ABB RAPID module: Module1.mod

MODULE Module1

     VAR robtarget current_position;
     VAR robtarget starting_position;
     VAR jointtarget joints;
    TASK PERS wobjdata wobj:=[FALSE,FALSE,"ROB_1",[[639.116,-22.796,-980.437],[1,0,0,0]],[[0,0,0],[1,0,0,0]]];

    PROC main()

starting_position := CRobT(\TaskName:="T_ROB1" \Tool:=Tooldata_9);
MoveJ RelTool (starting_position, 342,4, -480.2 \Rx:=7.6, \Ry:=21.9, \Rz:=1), v200, z200, Tooldata_9;
MoveJ RelTool (starting_position, 341,4, -481.5 \Rx:=7.6, \Ry:=21.6, \Rz:=1), v200, z200, Tooldata_9;
MoveJ RelTool (starting_position, 339,4, -483.2 \Rx:=7.6, \Ry:=21.6, \Rz:=1), v200, z200, Tooldata_9;
MoveJ RelTool (starting_position, 338,4, -485.4 \Rx:=7.5, \Ry:=21.3, \Rz:=1), v200, z200, Tooldata_9;
MoveJ RelTool (starting_position, 336,4, -488.1 \Rx:=7.5, \Ry:=21.3, \Rz:=1), v200, z200, Tooldata_9;
MoveJ RelTool (starting_position, 334,4, -491.4 \Rx:=7.5, \Ry:=21, \Rz:=1), v200, z200, Tooldata_9;
MoveJ RelTool (starting_position, 332,4, -495.2 \Rx:=7.5, \Ry:=20.7, \Rz:=1), v200, z200, Tooldata_9;
MoveJ RelTool (starting_position, 330,4, -499.5 \Rx:=7.5, \Ry:=20.4, \Rz:=1), v200, z200, Tooldata_9;
MoveJ RelTool (starting_position, 327,4, -504.2 \Rx:=7.5, \Ry:=20.1, \Rz:=1), v200, z200, Tooldata_9;
MoveJ RelTool (starting_position, 324,4, -509.1 \Rx:=7.5, \Ry:=19.8, \Rz:=1), v200, z200, Tooldata_9;
MoveJ RelTool (starting_position, 322,4, -514 \Rx:=7.6, \Ry:=19.5, \Rz:=1), v200, z200, Tooldata_9;
MoveJ RelTool (starting_position, 318,4, -518.8 \Rx:=7.6, \Ry:=19.5, \Rz:=1), v200, z200, Tooldata_9;
MoveJ RelTool (starting_position, 315,4, -523.4 \Rx:=7.6, \Ry:=19.2, \Rz:=1), v200, z200, Tooldata_9;
MoveJ RelTool (starting_position, 312,4, -527.5 \Rx:=7.6, \Ry:=18.9, \Rz:=1), v200, z200, Tooldata_9;
MoveJ RelTool (starting_position, 308,4, -531.3 \Rx:=7.6, \Ry:=18.6, \Rz:=1), v200, z200, Tooldata_9;
MoveJ RelTool (starting_position, 305,4, -534.7 \Rx:=7.6, \Ry:=18.3, \Rz:=1), v200, z200, Tooldata_9;
MoveJ RelTool (starting_position, 301,4, -537.8 \Rx:=7.6, \Ry:=18, \Rz:=1), v200, z200, Tooldata_9;
MoveJ RelTool (starting_position, 297,8, -540.6 \Rx:=7.6, \Ry:=17.4, \Rz:=2), v200, z200, Tooldata_9;
MoveJ RelTool (starting_position, 293,8, -543.1 \Rx:=7.6, \Ry:=17.1, \Rz:=2), v200, z200, Tooldata_9;
MoveJ RelTool (starting_position, 288,8, -545.5 \Rx:=7.6, \Ry:=16.8, \Rz:=2), v200, z200, Tooldata_9;
MoveJ RelTool (starting_position, 284,8, -547.8 \Rx:=7.6, \Ry:=16.5, \Rz:=2), v200, z200, Tooldata_9;
MoveJ RelTool (starting_position, 280,8, -550 \Rx:=7.6, \Ry:=15.9, \Rz:=2), v200, z200, Tooldata_9;
MoveJ RelTool (starting_position, 275,8, -552.2 \Rx:=7.6, \Ry:=15.6, \Rz:=2), v200, z200, Tooldata_9;
MoveJ RelTool (starting_position, 271,8, -554.4 \Rx:=7.6, \Ry:=15.3, \Rz:=2), v200, z200, Tooldata_9;
MoveJ RelTool (starting_position, 266,8, -556.6 \Rx:=7.7, \Ry:=14.7, \Rz:=2), v200, z200, Tooldata_9;
MoveJ RelTool (starting_position, 261,8, -558.8 \Rx:=7.7, \Ry:=14.4, \Rz:=2), v200, z200, Tooldata_9;
MoveJ RelTool (starting_position, 257,8, -561.1 \Rx:=7.7, \Ry:=14.1, \Rz:=2), v200, z200, Tooldata_9;
MoveJ RelTool (starting_position, 252,8, -563.3 \Rx:=7.7, \Ry:=13.5, \Rz:=2), v200, z200, Tooldata_9;
MoveJ RelTool (starting_position, 248,8, -565.6 \Rx:=7.7, \Ry:=13.2, \Rz:=2), v200, z200, Tooldata_9;
MoveJ RelTool (starting_position, 243,8, -567.8 \Rx:=7.7, \Ry:=12.9, \Rz:=2), v200, z200, Tooldata_9;
MoveJ RelTool (starting_position, 239,8, -570.1 \Rx:=7.7, \Ry:=12.3, \Rz:=2), v200, z200, Tooldata_9;
MoveJ RelTool (starting_position, 234,8, -572.3 \Rx:=7.7, \Ry:=12, \Rz:=2), v200, z200, Tooldata_9;
MoveJ RelTool (starting_position, 230,8, -574.4 \Rx:=7.7, \Ry:=11.7, \Rz:=2), v200, z200, Tooldata_9;
MoveJ RelTool (starting_position, 226,8, -576.4 \Rx:=7.7, \Ry:=11.4, \Rz:=2), v200, z200, Tooldata_9;
MoveJ RelTool (starting_position, 222,12, -578 \Rx:=7.8, \Ry:=10.8, \Rz:=3), v200, z200, Tooldata_9;
MoveJ RelTool (starting_position, 218,12, -579.3 \Rx:=7.8, \Ry:=10.5, \Rz:=3), v200, z200, Tooldata_9;
MoveJ RelTool (starting_position, 214,12, -580.4 \Rx:=7.8, \Ry:=10.2, \Rz:=3), v200, z200, Tooldata_9;
MoveJ RelTool (starting_position, 210,12, -581.1 \Rx:=7.8, \Ry:=9.9, \Rz:=3), v200, z200, Tooldata_9;
MoveJ RelTool (starting_position, 207,12, -581.4 \Rx:=7.8, \Ry:=9.6, \Rz:=3), v200, z200, Tooldata_9;
MoveJ RelTool (starting_position, 203,12, -581.5 \Rx:=7.8, \Ry:=9.3, \Rz:=3), v200, z200, Tooldata_9;
MoveJ RelTool (starting_position, 200,12, -581.3 \Rx:=7.8, \Ry:=9, \Rz:=3), v200, z200, Tooldata_9;
MoveJ RelTool (starting_position, 197,12, -580.9 \Rx:=7.8, \Ry:=8.7, \Rz:=3), v200, z200, Tooldata_9;
MoveJ RelTool (starting_position, 194,12, -580.4 \Rx:=7.8, \Ry:=8.4, \Rz:=3), v200, z200, Tooldata_9;
MoveJ RelTool (starting_position, 191,12, -579.7 \Rx:=7.8, \Ry:=8.4, \Rz:=3), v200, z200, Tooldata_9;
MoveJ RelTool (starting_position, 188,12, -579.2 \Rx:=7.8, \Ry:=8.1, \Rz:=3), v200, z200, Tooldata_9;
MoveJ RelTool (starting_position, 185,12, -578.8 \Rx:=7.8, \Ry:=7.8, \Rz:=3), v200, z200, Tooldata_9;
MoveJ RelTool (starting_position, 183,12, -578.9 \Rx:=7.8, \Ry:=7.5, \Rz:=3), v200, z200, Tooldata_9;
MoveJ RelTool (starting_position, 180,12, -579.4 \Rx:=7.8, \Ry:=7.2, \Rz:=3), v200, z200, Tooldata_9;
MoveJ RelTool (starting_position, 178,16, -580.4 \Rx:=7.8, \Ry:=7.2, \Rz:=4), v200, z200, Tooldata_9;
MoveJ RelTool (starting_position, 176,16, -582.1 \Rx:=7.8, \Ry:=6.9, \Rz:=4), v200, z200, Tooldata_9;
MoveJ RelTool (starting_position, 173,16, -584.3 \Rx:=7.8, \Ry:=6.9, \Rz:=4), v200, z200, Tooldata_9;
MoveJ RelTool (starting_position, 171,16, -587 \Rx:=7.8, \Ry:=6.6, \Rz:=4), v200, z200, Tooldata_9;
MoveJ RelTool (starting_position, 169,16, -589.9 \Rx:=7.8, \Ry:=6.3, \Rz:=4), v200, z200, Tooldata_9;
MoveJ RelTool (starting_position, 167,16, -592.9 \Rx:=7.8, \Ry:=6, \Rz:=4), v200, z200, Tooldata_9;
MoveJ RelTool (starting_position, 165,16, -595.7 \Rx:=7.7, \Ry:=6, \Rz:=4), v200, z200, Tooldata_9;
MoveJ RelTool (starting_position, 163,16, -598.3 \Rx:=7.7, \Ry:=6, \Rz:=4), v200, z200, Tooldata_9;
MoveJ RelTool (starting_position, 161,16, -600.4 \Rx:=7.7, \Ry:=5.7, \Rz:=4), v200, z200, Tooldata_9;
MoveJ RelTool (starting_position, 159,16, -602.1 \Rx:=7.7, \Ry:=5.4, \Rz:=4), v200, z200, Tooldata_9;
MoveJ RelTool (starting_position, 157,16, -603.5 \Rx:=7.7, \Ry:=5.4, \Rz:=4), v200, z200, Tooldata_9;
MoveJ RelTool (starting_position, 155,16, -604.4 \Rx:=7.6, \Ry:=5.1, \Rz:=4), v200, z200, Tooldata_9;
MoveJ RelTool (starting_position, 153,16, -605 \Rx:=7.6, \Ry:=5.1, \Rz:=4), v200, z200, Tooldata_9;
MoveJ RelTool (starting_position, 151,16, -605.4 \Rx:=7.6, \Ry:=4.8, \Rz:=4), v200, z200, Tooldata_9;
MoveJ RelTool (starting_position, 150,20, -605.6 \Rx:=7.5, \Ry:=4.8, \Rz:=5), v200, z200, Tooldata_9;
MoveJ RelTool (starting_position, 148,20, -605.7 \Rx:=7.5, \Ry:=4.5, \Rz:=5), v200, z200, Tooldata_9;
MoveJ RelTool (starting_position, 146,20, -605.8 \Rx:=7.5, \Ry:=4.5, \Rz:=5), v200, z200, Tooldata_9;
MoveJ RelTool (starting_position, 144,20, -605.8 \Rx:=7.4, \Ry:=4.2, \Rz:=5), v200, z200, Tooldata_9;
MoveJ RelTool (starting_position, 143,20, -605.8 \Rx:=7.4, \Ry:=4.2, \Rz:=5), v200, z200, Tooldata_9;
MoveJ RelTool (starting_position, 141,20, -605.8 \Rx:=7.3, \Ry:=3.9, \Rz:=5), v200, z200, Tooldata_9;
MoveJ RelTool (starting_position, 140,20, -605.8 \Rx:=7.3, \Ry:=3.9, \Rz:=5), v200, z200, Tooldata_9;
MoveJ RelTool (starting_position, 138,20, -605.8 \Rx:=7.2, \Ry:=3.6, \Rz:=5), v200, z200, Tooldata_9;
MoveJ RelTool (starting_position, 137,20, -605.8 \Rx:=7.2, \Ry:=3.6, \Rz:=5), v200, z200, Tooldata_9;
MoveJ RelTool (starting_position, 136,20, -605.8 \Rx:=7.1, \Ry:=3.6, \Rz:=5), v200, z200, Tooldata_9;
MoveJ RelTool (starting_position, 134,20, -605.8 \Rx:=7.1, \Ry:=3.3, \Rz:=5), v200, z200, Tooldata_9;
MoveJ RelTool (starting_position, 133,20, -605.8 \Rx:=7, \Ry:=3.3, \Rz:=5), v200, z200, Tooldata_9;
MoveJ RelTool (starting_position, 132,20, -605.8 \Rx:=6.9, \Ry:=3.3, \Rz:=5), v200, z200, Tooldata_9;
MoveJ RelTool (starting_position, 131,20, -605.8 \Rx:=6.9, \Ry:=3, \Rz:=5), v200, z200, Tooldata_9;
MoveJ RelTool (starting_position, 130,24, -605.8 \Rx:=6.8, \Ry:=3, \Rz:=6), v200, z200, Tooldata_9;
MoveJ RelTool (starting_position, 129,24, -605.8 \Rx:=6.7, \Ry:=3, \Rz:=6), v200, z200, Tooldata_9;
MoveJ RelTool (starting_position, 129,24, -605.8 \Rx:=6.7, \Ry:=3, \Rz:=6), v200, z200, Tooldata_9;
MoveJ RelTool (starting_position, 128,24, -605.8 \Rx:=6.6, \Ry:=2.7, \Rz:=6), v200, z200, Tooldata_9;
MoveJ RelTool (starting_position, 127,24, -606 \Rx:=6.5, \Ry:=2.7, \Rz:=6), v200, z200, Tooldata_9;
MoveJ RelTool (starting_position, 127,24, -606.4 \Rx:=6.4, \Ry:=2.7, \Rz:=6), v200, z200, Tooldata_9;
MoveJ RelTool (starting_position, 126,24, -606.9 \Rx:=6.3, \Ry:=2.7, \Rz:=6), v200, z200, Tooldata_9;
MoveJ RelTool (starting_position, 126,24, -607.5 \Rx:=6.2, \Ry:=2.7, \Rz:=6), v200, z200, Tooldata_9;
MoveJ RelTool (starting_position, 125,24, -608.2 \Rx:=6.2, \Ry:=2.7, \Rz:=6), v200, z200, Tooldata_9;
MoveJ RelTool (starting_position, 125,24, -609.1 \Rx:=6.1, \Ry:=2.7, \Rz:=6), v200, z200, Tooldata_9;
MoveJ RelTool (starting_position, 124,24, -610.2 \Rx:=6, \Ry:=2.7, \Rz:=6), v200, z200, Tooldata_9;
MoveJ RelTool (starting_position, 123,24, -611.3 \Rx:=5.9, \Ry:=2.4, \Rz:=6), v200, z200, Tooldata_9;
MoveJ RelTool (starting_position, 123,24, -612.3 \Rx:=5.8, \Ry:=2.4, \Rz:=6), v200, z200, Tooldata_9;
MoveJ RelTool (starting_position, 122,24, -613.3 \Rx:=5.7, \Ry:=2.4, \Rz:=6), v200, z200, Tooldata_9;
MoveJ RelTool (starting_position, 121,28, -614.1 \Rx:=5.7, \Ry:=2.4, \Rz:=7), v200, z200, Tooldata_9;
MoveJ RelTool (starting_position, 120,28, -614.8 \Rx:=5.6, \Ry:=2.1, \Rz:=7), v200, z200, Tooldata_9;
MoveJ RelTool (starting_position, 119,28, -615.4 \Rx:=5.5, \Ry:=2.1, \Rz:=7), v200, z200, Tooldata_9;
MoveJ RelTool (starting_position, 118,28, -616 \Rx:=5.4, \Ry:=2.1, \Rz:=7), v200, z200, Tooldata_9;
MoveJ RelTool (starting_position, 117,28, -616.7 \Rx:=5.3, \Ry:=1.8, \Rz:=7), v200, z200, Tooldata_9;
MoveJ RelTool (starting_position, 117,28, -617.3 \Rx:=5.3, \Ry:=1.8, \Rz:=7), v200, z200, Tooldata_9;
MoveJ RelTool (starting_position, 116,28, -618 \Rx:=5.2, \Ry:=1.8, \Rz:=7), v200, z200, Tooldata_9;
MoveJ RelTool (starting_position, 115,28, -618.7 \Rx:=5.1, \Ry:=1.8, \Rz:=7), v200, z200, Tooldata_9;
MoveJ RelTool (starting_position, 114,28, -619.2 \Rx:=5, \Ry:=1.8, \Rz:=7), v200, z200, Tooldata_9;
MoveJ RelTool (starting_position, 113,28, -619.6 \Rx:=4.9, \Ry:=1.5, \Rz:=7), v200, z200, Tooldata_9;
MoveJ RelTool (starting_position, 112,28, -619.8 \Rx:=4.8, \Ry:=1.5, \Rz:=7), v200, z200, Tooldata_9;
MoveJ RelTool (starting_position, 112,28, -619.9 \Rx:=4.7, \Ry:=1.5, \Rz:=7), v200, z200, Tooldata_9;
MoveJ RelTool (starting_position, 111,28, -619.8 \Rx:=4.6, \Ry:=1.5, \Rz:=7), v200, z200, Tooldata_9;
MoveJ RelTool (starting_position, 110,28, -619.5 \Rx:=4.5, \Ry:=1.2, \Rz:=7), v200, z200, Tooldata_9;
MoveJ RelTool (starting_position, 109,28, -619.2 \Rx:=4.4, \Ry:=1.2, \Rz:=7), v200, z200, Tooldata_9;
MoveJ RelTool (starting_position, 108,28, -618.8 \Rx:=4.4, \Ry:=1.2, \Rz:=7), v200, z200, Tooldata_9;
MoveJ RelTool (starting_position, 107,32, -618.4 \Rx:=4.3, \Ry:=1.2, \Rz:=8), v200, z200, Tooldata_9;
MoveJ RelTool (starting_position, 107,32, -618.2 \Rx:=4.2, \Ry:=0.9, \Rz:=8), v200, z200, Tooldata_9;
MoveJ RelTool (starting_position, 106,32, -618.1 \Rx:=4.1, \Ry:=0.9, \Rz:=8), v200, z200, Tooldata_9;
MoveJ RelTool (starting_position, 105,32, -618.2 \Rx:=4, \Ry:=0.9, \Rz:=8), v200, z200, Tooldata_9;
MoveJ RelTool (starting_position, 104,32, -618.4 \Rx:=3.9, \Ry:=0.9, \Rz:=8), v200, z200, Tooldata_9;
MoveJ RelTool (starting_position, 103,32, -618.8 \Rx:=3.8, \Ry:=0.6, \Rz:=8), v200, z200, Tooldata_9;
MoveJ RelTool (starting_position, 102,32, -619.2 \Rx:=3.7, \Ry:=0.6, \Rz:=8), v200, z200, Tooldata_9;
MoveJ RelTool (starting_position, 102,32, -619.7 \Rx:=3.6, \Ry:=0.6, \Rz:=8), v200, z200, Tooldata_9;
MoveJ RelTool (starting_position, 101,32, -620.1 \Rx:=3.6, \Ry:=0.6, \Rz:=8), v200, z200, Tooldata_9;
MoveJ RelTool (starting_position, 100,32, -620.4 \Rx:=3.5, \Ry:=0.6, \Rz:=8), v200, z200, Tooldata_9;
MoveJ RelTool (starting_position, 99,32, -620.7 \Rx:=3.4, \Ry:=0.3, \Rz:=8), v200, z200, Tooldata_9;
MoveJ RelTool (starting_position, 99,32, -620.8 \Rx:=3.3, \Ry:=0.3, \Rz:=8), v200, z200, Tooldata_9;
MoveJ RelTool (starting_position, 98,32, -620.9 \Rx:=3.2, \Ry:=0.3, \Rz:=8), v200, z200, Tooldata_9;
MoveJ RelTool (starting_position, 97,32, -620.9 \Rx:=3.2, \Ry:=0.3, \Rz:=8), v200, z200, Tooldata_9;
MoveJ RelTool (starting_position, 96,32, -620.7 \Rx:=3.1, \Ry:=0, \Rz:=8), v200, z200, Tooldata_9;
MoveJ RelTool (starting_position, 95,36, -620.5 \Rx:=3, \Ry:=0, \Rz:=9), v200, z200, Tooldata_9;
MoveJ RelTool (starting_position, 94,36, -620.2 \Rx:=2.9, \Ry:=-0, \Rz:=9), v200, z200, Tooldata_9;
MoveJ RelTool (starting_position, 94,36, -619.8 \Rx:=2.9, \Ry:=-0, \Rz:=9), v200, z200, Tooldata_9;
MoveJ RelTool (starting_position, 93,36, -619.4 \Rx:=2.8, \Ry:=-0.3, \Rz:=9), v200, z200, Tooldata_9;
MoveJ RelTool (starting_position, 92,36, -619 \Rx:=2.7, \Ry:=-0.3, \Rz:=9), v200, z200, Tooldata_9;
MoveJ RelTool (starting_position, 91,36, -618.5 \Rx:=2.7, \Ry:=-0.3, \Rz:=9), v200, z200, Tooldata_9;
MoveJ RelTool (starting_position, 90,36, -618.2 \Rx:=2.6, \Ry:=-0.3, \Rz:=9), v200, z200, Tooldata_9;
MoveJ RelTool (starting_position, 90,36, -617.9 \Rx:=2.5, \Ry:=-0.6, \Rz:=9), v200, z200, Tooldata_9;
MoveJ RelTool (starting_position, 89,36, -617.7 \Rx:=2.4, \Ry:=-0.6, \Rz:=9), v200, z200, Tooldata_9;
MoveJ RelTool (starting_position, 88,36, -617.7 \Rx:=2.4, \Ry:=-0.6, \Rz:=9), v200, z200, Tooldata_9;
MoveJ RelTool (starting_position, 87,36, -617.7 \Rx:=2.3, \Ry:=-0.6, \Rz:=9), v200, z200, Tooldata_9;
MoveJ RelTool (starting_position, 86,36, -617.8 \Rx:=2.2, \Ry:=-0.6, \Rz:=9), v200, z200, Tooldata_9;
MoveJ RelTool (starting_position, 85,36, -617.9 \Rx:=2.2, \Ry:=-0.6, \Rz:=9), v200, z200, Tooldata_9;
MoveJ RelTool (starting_position, 84,36, -618 \Rx:=2.1, \Ry:=-0.9, \Rz:=9), v200, z200, Tooldata_9;
MoveJ RelTool (starting_position, 83,36, -618.1 \Rx:=2, \Ry:=-0.9, \Rz:=9), v200, z200, Tooldata_9;
MoveJ RelTool (starting_position, 81,36, -618.1 \Rx:=1.9, \Ry:=-1.2, \Rz:=9), v200, z200, Tooldata_9;
MoveJ RelTool (starting_position, 80,36, -618.2 \Rx:=1.9, \Ry:=-1.2, \Rz:=9), v200, z200, Tooldata_9;
MoveJ RelTool (starting_position, 78,40, -618.2 \Rx:=1.8, \Ry:=-1.5, \Rz:=10), v200, z200, Tooldata_9;
MoveJ RelTool (starting_position, 77,40, -618.3 \Rx:=1.7, \Ry:=-1.5, \Rz:=10), v200, z200, Tooldata_9;
MoveJ RelTool (starting_position, 75,40, -618.3 \Rx:=1.7, \Ry:=-1.5, \Rz:=10), v200, z200, Tooldata_9;
MoveJ RelTool (starting_position, 73,40, -618.3 \Rx:=1.6, \Ry:=-1.8, \Rz:=10), v200, z200, Tooldata_9;
MoveJ RelTool (starting_position, 72,40, -618.3 \Rx:=1.6, \Ry:=-2.1, \Rz:=10), v200, z200, Tooldata_9;
MoveJ RelTool (starting_position, 70,40, -618.3 \Rx:=1.5, \Ry:=-2.1, \Rz:=10), v200, z200, Tooldata_9;
MoveJ RelTool (starting_position, 68,40, -618.3 \Rx:=1.4, \Ry:=-2.4, \Rz:=10), v200, z200, Tooldata_9;
MoveJ RelTool (starting_position, 66,40, -618.3 \Rx:=1.4, \Ry:=-2.4, \Rz:=10), v200, z200, Tooldata_9;
MoveJ RelTool (starting_position, 65,40, -618.3 \Rx:=1.3, \Ry:=-2.7, \Rz:=10), v200, z200, Tooldata_9;
MoveJ RelTool (starting_position, 63,40, -618.3 \Rx:=1.3, \Ry:=-2.7, \Rz:=10), v200, z200, Tooldata_9;
MoveJ RelTool (starting_position, 61,40, -618.3 \Rx:=1.2, \Ry:=-3, \Rz:=10), v200, z200, Tooldata_9;
MoveJ RelTool (starting_position, 59,40, -618.3 \Rx:=1.2, \Ry:=-3, \Rz:=10), v200, z200, Tooldata_9;
MoveJ RelTool (starting_position, 57,40, -618.3 \Rx:=1.1, \Ry:=-3.3, \Rz:=10), v200, z200, Tooldata_9;
MoveJ RelTool (starting_position, 56,40, -618.2 \Rx:=1.1, \Ry:=-3.3, \Rz:=10), v200, z200, Tooldata_9;
MoveJ RelTool (starting_position, 54,40, -618 \Rx:=1, \Ry:=-3.6, \Rz:=10), v200, z200, Tooldata_9;
MoveJ RelTool (starting_position, 52,40, -617.8 \Rx:=0.9, \Ry:=-3.6, \Rz:=10), v200, z200, Tooldata_9;
MoveJ RelTool (starting_position, 50,40, -617.3 \Rx:=0.9, \Ry:=-3.9, \Rz:=10), v200, z200, Tooldata_9;
MoveJ RelTool (starting_position, 49,40, -616.7 \Rx:=0.8, \Ry:=-4.2, \Rz:=10), v200, z200, Tooldata_9;
MoveJ RelTool (starting_position, 47,44, -615.8 \Rx:=0.8, \Ry:=-4.2, \Rz:=11), v200, z200, Tooldata_9;
MoveJ RelTool (starting_position, 46,44, -614.7 \Rx:=0.7, \Ry:=-4.2, \Rz:=11), v200, z200, Tooldata_9;
MoveJ RelTool (starting_position, 44,44, -613.4 \Rx:=0.7, \Ry:=-4.5, \Rz:=11), v200, z200, Tooldata_9;
MoveJ RelTool (starting_position, 43,44, -611.8 \Rx:=0.6, \Ry:=-4.5, \Rz:=11), v200, z200, Tooldata_9;
MoveJ RelTool (starting_position, 42,44, -610.2 \Rx:=0.5, \Ry:=-4.8, \Rz:=11), v200, z200, Tooldata_9;
MoveJ RelTool (starting_position, 41,44, -608.5 \Rx:=0.5, \Ry:=-4.8, \Rz:=11), v200, z200, Tooldata_9;
MoveJ RelTool (starting_position, 40,44, -607 \Rx:=0.4, \Ry:=-4.8, \Rz:=11), v200, z200, Tooldata_9;
MoveJ RelTool (starting_position, 39,44, -605.6 \Rx:=0.4, \Ry:=-4.8, \Rz:=11), v200, z200, Tooldata_9;
MoveJ RelTool (starting_position, 38,44, -604.4 \Rx:=0.3, \Ry:=-5.1, \Rz:=11), v200, z200, Tooldata_9;
MoveJ RelTool (starting_position, 38,44, -603.5 \Rx:=0.3, \Ry:=-5.1, \Rz:=11), v200, z200, Tooldata_9;
MoveJ RelTool (starting_position, 38,44, -602.9 \Rx:=0.2, \Ry:=-5.1, \Rz:=11), v200, z200, Tooldata_9;
MoveJ RelTool (starting_position, 38,44, -602.3 \Rx:=0.2, \Ry:=-5.1, \Rz:=11), v200, z200, Tooldata_9;
MoveJ RelTool (starting_position, 38,44, -601.9 \Rx:=0.1, \Ry:=-5.1, \Rz:=11), v200, z200, Tooldata_9;
MoveJ RelTool (starting_position, 38,44, -601.4 \Rx:=0.1, \Ry:=-5.1, \Rz:=11), v200, z200, Tooldata_9;
MoveJ RelTool (starting_position, 39,44, -600.8 \Rx:=0, \Ry:=-4.8, \Rz:=11), v200, z200, Tooldata_9;
MoveJ RelTool (starting_position, 40,44, -600.2 \Rx:=-0, \Ry:=-4.8, \Rz:=11), v200, z200, Tooldata_9;
MoveJ RelTool (starting_position, 41,44, -599.3 \Rx:=-0.1, \Ry:=-4.8, \Rz:=11), v200, z200, Tooldata_9;
MoveJ RelTool (starting_position, 42,44, -598.1 \Rx:=-0.1, \Ry:=-4.5, \Rz:=11), v200, z200, Tooldata_9;
MoveJ RelTool (starting_position, 44,44, -596.6 \Rx:=-0.2, \Ry:=-4.5, \Rz:=11), v200, z200, Tooldata_9;
MoveJ RelTool (starting_position, 45,44, -594.9 \Rx:=-0.2, \Ry:=-4.5, \Rz:=11), v200, z200, Tooldata_9;
MoveJ RelTool (starting_position, 47,48, -593.1 \Rx:=-0.3, \Ry:=-4.2, \Rz:=12), v200, z200, Tooldata_9;
MoveJ RelTool (starting_position, 48,48, -591 \Rx:=-0.3, \Ry:=-4.2, \Rz:=12), v200, z200, Tooldata_9;
MoveJ RelTool (starting_position, 50,48, -589 \Rx:=-0.4, \Ry:=-3.9, \Rz:=12), v200, z200, Tooldata_9;
MoveJ RelTool (starting_position, 52,48, -587 \Rx:=-0.4, \Ry:=-3.6, \Rz:=12), v200, z200, Tooldata_9;
MoveJ RelTool (starting_position, 55,48, -585.3 \Rx:=-0.4, \Ry:=-3.6, \Rz:=12), v200, z200, Tooldata_9;
MoveJ RelTool (starting_position, 57,48, -583.8 \Rx:=-0.5, \Ry:=-3.3, \Rz:=12), v200, z200, Tooldata_9;
MoveJ RelTool (starting_position, 59,48, -582.7 \Rx:=-0.5, \Ry:=-3, \Rz:=12), v200, z200, Tooldata_9;
MoveJ RelTool (starting_position, 61,48, -582 \Rx:=-0.6, \Ry:=-3, \Rz:=12), v200, z200, Tooldata_9;
MoveJ RelTool (starting_position, 64,48, -581.6 \Rx:=-0.6, \Ry:=-2.7, \Rz:=12), v200, z200, Tooldata_9;
MoveJ RelTool (starting_position, 66,48, -581.8 \Rx:=-0.7, \Ry:=-2.4, \Rz:=12), v200, z200, Tooldata_9;
MoveJ RelTool (starting_position, 68,48, -582.3 \Rx:=-0.7, \Ry:=-2.4, \Rz:=12), v200, z200, Tooldata_9;
MoveJ RelTool (starting_position, 71,48, -583.1 \Rx:=-0.7, \Ry:=-2.1, \Rz:=12), v200, z200, Tooldata_9;
MoveJ RelTool (starting_position, 73,48, -584.2 \Rx:=-0.8, \Ry:=-1.8, \Rz:=12), v200, z200, Tooldata_9;
MoveJ RelTool (starting_position, 75,48, -585.4 \Rx:=-0.8, \Ry:=-1.5, \Rz:=12), v200, z200, Tooldata_9;
MoveJ RelTool (starting_position, 77,48, -586.5 \Rx:=-0.8, \Ry:=-1.5, \Rz:=12), v200, z200, Tooldata_9;
MoveJ RelTool (starting_position, 79,48, -587.5 \Rx:=-0.9, \Ry:=-1.2, \Rz:=12), v200, z200, Tooldata_9;
MoveJ RelTool (starting_position, 81,48, -588.4 \Rx:=-0.9, \Ry:=-1.2, \Rz:=12), v200, z200, Tooldata_9;
MoveJ RelTool (starting_position, 83,48, -589 \Rx:=-1, \Ry:=-0.9, \Rz:=12), v200, z200, Tooldata_9;
MoveJ RelTool (starting_position, 85,48, -589.4 \Rx:=-1, \Ry:=-0.9, \Rz:=12), v200, z200, Tooldata_9;
MoveJ RelTool (starting_position, 86,48, -589.6 \Rx:=-1, \Ry:=-0.6, \Rz:=12), v200, z200, Tooldata_9;
MoveJ RelTool (starting_position, 88,48, -589.7 \Rx:=-1.1, \Ry:=-0.6, \Rz:=12), v200, z200, Tooldata_9;
MoveJ RelTool (starting_position, 90,48, -589.6 \Rx:=-1.1, \Ry:=-0.3, \Rz:=12), v200, z200, Tooldata_9;
MoveJ RelTool (starting_position, 91,52, -589.6 \Rx:=-1.1, \Ry:=-0.3, \Rz:=13), v200, z200, Tooldata_9;
MoveJ RelTool (starting_position, 92,52, -589.5 \Rx:=-1.2, \Ry:=-0, \Rz:=13), v200, z200, Tooldata_9;
MoveJ RelTool (starting_position, 94,52, -589.5 \Rx:=-1.2, \Ry:=0, \Rz:=13), v200, z200, Tooldata_9;
MoveJ RelTool (starting_position, 95,52, -589.6 \Rx:=-1.2, \Ry:=0, \Rz:=13), v200, z200, Tooldata_9;
MoveJ RelTool (starting_position, 96,52, -589.8 \Rx:=-1.3, \Ry:=0, \Rz:=13), v200, z200, Tooldata_9;
MoveJ RelTool (starting_position, 97,52, -590 \Rx:=-1.3, \Ry:=0.3, \Rz:=13), v200, z200, Tooldata_9;
MoveJ RelTool (starting_position, 98,52, -590.2 \Rx:=-1.3, \Ry:=0.3, \Rz:=13), v200, z200, Tooldata_9;
MoveJ RelTool (starting_position, 98,52, -590.4 \Rx:=-1.3, \Ry:=0.3, \Rz:=13), v200, z200, Tooldata_9;
MoveJ RelTool (starting_position, 99,52, -590.5 \Rx:=-1.4, \Ry:=0.6, \Rz:=13), v200, z200, Tooldata_9;
MoveJ RelTool (starting_position, 100,52, -590.6 \Rx:=-1.4, \Ry:=0.3, \Rz:=13), v200, z200, Tooldata_9;
MoveJ RelTool (starting_position, 100,52, -590.7 \Rx:=-1.4, \Ry:=0.6, \Rz:=13), v200, z200, Tooldata_9;
MoveJ RelTool (starting_position, 101,52, -590.8 \Rx:=-1.4, \Ry:=0.6, \Rz:=13), v200, z200, Tooldata_9;
MoveJ RelTool (starting_position, 101,52, -590.9 \Rx:=-1.4, \Ry:=0.6, \Rz:=13), v200, z200, Tooldata_9;
MoveJ RelTool (starting_position, 102,52, -590.9 \Rx:=-1.4, \Ry:=0.6, \Rz:=13), v200, z200, Tooldata_9;
MoveJ RelTool (starting_position, 102,52, -590.9 \Rx:=-1.4, \Ry:=0.6, \Rz:=13), v200, z200, Tooldata_9;
MoveJ RelTool (starting_position, 102,52, -590.9 \Rx:=-1.4, \Ry:=0.6, \Rz:=13), v200, z200, Tooldata_9;
MoveJ RelTool (starting_position, 103,52, -590.9 \Rx:=-1.4, \Ry:=0.6, \Rz:=13), v200, z200, Tooldata_9;
MoveJ RelTool (starting_position, 103,52, -590.9 \Rx:=-1.4, \Ry:=0.6, \Rz:=13), v200, z200, Tooldata_9;
MoveJ RelTool (starting_position, 104,52, -590.9 \Rx:=-1.4, \Ry:=0.9, \Rz:=13), v200, z200, Tooldata_9;
MoveJ RelTool (starting_position, 105,52, -590.9 \Rx:=-1.4, \Ry:=0.9, \Rz:=13), v200, z200, Tooldata_9;
MoveJ RelTool (starting_position, 105,52, -590.9 \Rx:=-1.4, \Ry:=0.9, \Rz:=13), v200, z200, Tooldata_9;
MoveJ RelTool (starting_position, 106,52, -590.9 \Rx:=-1.4, \Ry:=0.9, \Rz:=13), v200, z200, Tooldata_9;
MoveJ RelTool (starting_position, 107,52, -590.9 \Rx:=-1.4, \Ry:=0.9, \Rz:=13), v200, z200, Tooldata_9;
MoveJ RelTool (starting_position, 108,52, -590.9 \Rx:=-1.4, \Ry:=1.2, \Rz:=13), v200, z200, Tooldata_9;
MoveJ RelTool (starting_position, 109,52, -590.9 \Rx:=-1.4, \Ry:=1.2, \Rz:=13), v200, z200, Tooldata_9;
MoveJ RelTool (starting_position, 110,52, -590.9 \Rx:=-1.4, \Ry:=1.5, \Rz:=13), v200, z200, Tooldata_9;
MoveJ RelTool (starting_position, 111,52, -590.9 \Rx:=-1.4, \Ry:=1.2, \Rz:=13), v200, z200, Tooldata_9;
MoveJ RelTool (starting_position, 112,56, -590.9 \Rx:=-1.4, \Ry:=1.5, \Rz:=14), v200, z200, Tooldata_9;
MoveJ RelTool (starting_position, 113,56, -590.9 \Rx:=-1.4, \Ry:=1.5, \Rz:=14), v200, z200, Tooldata_9;
MoveJ RelTool (starting_position, 115,56, -590.9 \Rx:=-1.4, \Ry:=1.8, \Rz:=14), v200, z200, Tooldata_9;
MoveJ RelTool (starting_position, 116,56, -590.9 \Rx:=-1.3, \Ry:=1.8, \Rz:=14), v200, z200, Tooldata_9;
MoveJ RelTool (starting_position, 117,56, -590.9 \Rx:=-1.3, \Ry:=1.8, \Rz:=14), v200, z200, Tooldata_9;
MoveJ RelTool (starting_position, 119,56, -590.9 \Rx:=-1.3, \Ry:=2.1, \Rz:=14), v200, z200, Tooldata_9;
MoveJ RelTool (starting_position, 120,56, -590.9 \Rx:=-1.3, \Ry:=2.1, \Rz:=14), v200, z200, Tooldata_9;
MoveJ RelTool (starting_position, 121,56, -590.8 \Rx:=-1.3, \Ry:=2.4, \Rz:=14), v200, z200, Tooldata_9;
MoveJ RelTool (starting_position, 123,56, -590.7 \Rx:=-1.2, \Ry:=2.4, \Rz:=14), v200, z200, Tooldata_9;
MoveJ RelTool (starting_position, 124,56, -590.6 \Rx:=-1.2, \Ry:=2.7, \Rz:=14), v200, z200, Tooldata_9;
MoveJ RelTool (starting_position, 126,56, -590.6 \Rx:=-1.2, \Ry:=2.7, \Rz:=14), v200, z200, Tooldata_9;
MoveJ RelTool (starting_position, 127,56, -590.6 \Rx:=-1.1, \Ry:=2.7, \Rz:=14), v200, z200, Tooldata_9;
MoveJ RelTool (starting_position, 128,56, -590.6 \Rx:=-1.1, \Ry:=3, \Rz:=14), v200, z200, Tooldata_9;
MoveJ RelTool (starting_position, 130,56, -590.7 \Rx:=-1.1, \Ry:=3, \Rz:=14), v200, z200, Tooldata_9;
MoveJ RelTool (starting_position, 131,56, -591 \Rx:=-1.1, \Ry:=3.3, \Rz:=14), v200, z200, Tooldata_9;
MoveJ RelTool (starting_position, 132,56, -591.5 \Rx:=-1, \Ry:=3.3, \Rz:=14), v200, z200, Tooldata_9;
MoveJ RelTool (starting_position, 133,56, -592.2 \Rx:=-1, \Ry:=3.3, \Rz:=14), v200, z200, Tooldata_9;
MoveJ RelTool (starting_position, 134,56, -593.2 \Rx:=-1, \Ry:=3.3, \Rz:=14), v200, z200, Tooldata_9;
MoveJ RelTool (starting_position, 134,56, -594.3 \Rx:=-0.9, \Ry:=3.6, \Rz:=14), v200, z200, Tooldata_9;
MoveJ RelTool (starting_position, 135,56, -595.6 \Rx:=-0.9, \Ry:=3.6, \Rz:=14), v200, z200, Tooldata_9;
MoveJ RelTool (starting_position, 136,56, -597 \Rx:=-0.8, \Ry:=3.6, \Rz:=14), v200, z200, Tooldata_9;
MoveJ RelTool (starting_position, 136,56, -598.3 \Rx:=-0.8, \Ry:=3.6, \Rz:=14), v200, z200, Tooldata_9;
MoveJ RelTool (starting_position, 136,56, -599.6 \Rx:=-0.7, \Ry:=3.9, \Rz:=14), v200, z200, Tooldata_9;
MoveJ RelTool (starting_position, 136,56, -600.7 \Rx:=-0.7, \Ry:=3.6, \Rz:=14), v200, z200, Tooldata_9;
MoveJ RelTool (starting_position, 136,56, -601.6 \Rx:=-0.6, \Ry:=3.6, \Rz:=14), v200, z200, Tooldata_9;
MoveJ RelTool (starting_position, 136,56, -602.4 \Rx:=-0.6, \Ry:=3.9, \Rz:=14), v200, z200, Tooldata_9;
MoveJ RelTool (starting_position, 136,56, -603 \Rx:=-0.5, \Ry:=3.6, \Rz:=14), v200, z200, Tooldata_9;
MoveJ RelTool (starting_position, 135,56, -603.6 \Rx:=-0.4, \Ry:=3.6, \Rz:=14), v200, z200, Tooldata_9;
MoveJ RelTool (starting_position, 134,56, -604.2 \Rx:=-0.4, \Ry:=3.6, \Rz:=14), v200, z200, Tooldata_9;
MoveJ RelTool (starting_position, 133,56, -604.7 \Rx:=-0.3, \Ry:=3.3, \Rz:=14), v200, z200, Tooldata_9;
MoveJ RelTool (starting_position, 132,56, -605.3 \Rx:=-0.2, \Ry:=3.3, \Rz:=14), v200, z200, Tooldata_9;
MoveJ RelTool (starting_position, 131,56, -606 \Rx:=-0.2, \Ry:=3.3, \Rz:=14), v200, z200, Tooldata_9;
MoveJ RelTool (starting_position, 130,56, -606.9 \Rx:=-0.1, \Ry:=3, \Rz:=14), v200, z200, Tooldata_9;
MoveJ RelTool (starting_position, 128,56, -608 \Rx:=-0.1, \Ry:=3, \Rz:=14), v200, z200, Tooldata_9;
MoveJ RelTool (starting_position, 126,56, -609.3 \Rx:=0, \Ry:=2.7, \Rz:=14), v200, z200, Tooldata_9;
MoveJ RelTool (starting_position, 125,56, -610.8 \Rx:=0.1, \Ry:=2.7, \Rz:=14), v200, z200, Tooldata_9;
MoveJ RelTool (starting_position, 123,56, -612.4 \Rx:=0.1, \Ry:=2.4, \Rz:=14), v200, z200, Tooldata_9;
MoveJ RelTool (starting_position, 121,56, -614 \Rx:=0.2, \Ry:=2.4, \Rz:=14), v200, z200, Tooldata_9;
MoveJ RelTool (starting_position, 118,60, -615.6 \Rx:=0.3, \Ry:=2.1, \Rz:=15), v200, z200, Tooldata_9;
MoveJ RelTool (starting_position, 116,60, -617.1 \Rx:=0.4, \Ry:=2.1, \Rz:=15), v200, z200, Tooldata_9;
MoveJ RelTool (starting_position, 113,60, -618.4 \Rx:=0.4, \Ry:=1.8, \Rz:=15), v200, z200, Tooldata_9;
MoveJ RelTool (starting_position, 111,60, -619.5 \Rx:=0.5, \Ry:=1.5, \Rz:=15), v200, z200, Tooldata_9;
MoveJ RelTool (starting_position, 108,60, -620.3 \Rx:=0.5, \Ry:=1.2, \Rz:=15), v200, z200, Tooldata_9;
MoveJ RelTool (starting_position, 105,60, -620.8 \Rx:=0.6, \Ry:=0.9, \Rz:=15), v200, z200, Tooldata_9;
MoveJ RelTool (starting_position, 101,60, -621 \Rx:=0.6, \Ry:=0.6, \Rz:=15), v200, z200, Tooldata_9;
MoveJ RelTool (starting_position, 98,60, -620.8 \Rx:=0.7, \Ry:=0.3, \Rz:=15), v200, z200, Tooldata_9;
MoveJ RelTool (starting_position, 95,60, -620.3 \Rx:=0.7, \Ry:=0, \Rz:=15), v200, z200, Tooldata_9;
MoveJ RelTool (starting_position, 91,60, -619.4 \Rx:=0.8, \Ry:=-0.3, \Rz:=15), v200, z200, Tooldata_9;
MoveJ RelTool (starting_position, 88,60, -618.2 \Rx:=0.8, \Ry:=-0.6, \Rz:=15), v200, z200, Tooldata_9;
MoveJ RelTool (starting_position, 84,60, -616.7 \Rx:=0.9, \Ry:=-0.9, \Rz:=15), v200, z200, Tooldata_9;
MoveJ RelTool (starting_position, 80,60, -615.1 \Rx:=0.9, \Ry:=-1.2, \Rz:=15), v200, z200, Tooldata_9;
MoveJ RelTool (starting_position, 77,60, -613.4 \Rx:=1, \Ry:=-1.5, \Rz:=15), v200, z200, Tooldata_9;
MoveJ RelTool (starting_position, 73,60, -611.7 \Rx:=1.1, \Ry:=-1.8, \Rz:=15), v200, z200, Tooldata_9;
MoveJ RelTool (starting_position, 69,60, -610 \Rx:=1.1, \Ry:=-2.1, \Rz:=15), v200, z200, Tooldata_9;
MoveJ RelTool (starting_position, 64,60, -608.3 \Rx:=1.2, \Ry:=-2.7, \Rz:=15), v200, z200, Tooldata_9;
MoveJ RelTool (starting_position, 60,60, -606.8 \Rx:=1.2, \Ry:=-3, \Rz:=15), v200, z200, Tooldata_9;
MoveJ RelTool (starting_position, 56,60, -605.4 \Rx:=1.3, \Ry:=-3.3, \Rz:=15), v200, z200, Tooldata_9;
MoveJ RelTool (starting_position, 51,60, -604.3 \Rx:=1.3, \Ry:=-3.6, \Rz:=15), v200, z200, Tooldata_9;
MoveJ RelTool (starting_position, 46,60, -603.5 \Rx:=1.4, \Ry:=-3.9, \Rz:=15), v200, z200, Tooldata_9;
MoveJ RelTool (starting_position, 41,60, -603.1 \Rx:=1.5, \Ry:=-4.5, \Rz:=15), v200, z200, Tooldata_9;
MoveJ RelTool (starting_position, 35,60, -603.2 \Rx:=1.5, \Ry:=-5.1, \Rz:=15), v200, z200, Tooldata_9;
MoveJ RelTool (starting_position, 30,60, -603.5 \Rx:=1.6, \Ry:=-5.7, \Rz:=15), v200, z200, Tooldata_9;
MoveJ RelTool (starting_position, 24,60, -604.1 \Rx:=1.6, \Ry:=-6, \Rz:=15), v200, z200, Tooldata_9;
MoveJ RelTool (starting_position, 18,60, -604.9 \Rx:=1.7, \Ry:=-6.3, \Rz:=15), v200, z200, Tooldata_9;
MoveJ RelTool (starting_position, 12,60, -605.8 \Rx:=1.7, \Ry:=-7.2, \Rz:=15), v200, z200, Tooldata_9;
MoveJ RelTool (starting_position, 6,60, -606.5 \Rx:=1.7, \Ry:=-7.8, \Rz:=15), v200, z200, Tooldata_9;
MoveJ RelTool (starting_position, 0,60, -607.1 \Rx:=1.7, \Ry:=-8.1, \Rz:=15), v200, z200, Tooldata_9;
MoveJ RelTool (starting_position, -7,60, -607.5 \Rx:=1.7, \Ry:=-8.7, \Rz:=15), v200, z200, Tooldata_9;
MoveJ RelTool (starting_position, -13,60, -607.8 \Rx:=1.8, \Ry:=-9.3, \Rz:=15), v200, z200, Tooldata_9;
MoveJ RelTool (starting_position, -20,60, -608.2 \Rx:=1.8, \Ry:=-9.9, \Rz:=15), v200, z200, Tooldata_9;
MoveJ RelTool (starting_position, -27,60, -608.7 \Rx:=1.9, \Ry:=-10.5, \Rz:=15), v200, z200, Tooldata_9;
MoveJ RelTool (starting_position, -33,60, -609.3 \Rx:=1.9, \Ry:=-11.1, \Rz:=15), v200, z200, Tooldata_9;
MoveJ RelTool (starting_position, -40,60, -610 \Rx:=1.9, \Ry:=-11.7, \Rz:=15), v200, z200, Tooldata_9;
MoveJ RelTool (starting_position, -46,60, -610.9 \Rx:=1.9, \Ry:=-12.3, \Rz:=15), v200, z200, Tooldata_9;
MoveJ RelTool (starting_position, -53,60, -611.8 \Rx:=1.9, \Ry:=-12.9, \Rz:=15), v200, z200, Tooldata_9;
MoveJ RelTool (starting_position, -59,60, -612.6 \Rx:=1.9, \Ry:=-13.5, \Rz:=15), v200, z200, Tooldata_9;
MoveJ RelTool (starting_position, -65,60, -613 \Rx:=1.9, \Ry:=-14.1, \Rz:=15), v200, z200, Tooldata_9;
MoveJ RelTool (starting_position, -70,60, -613 \Rx:=1.9, \Ry:=-14.7, \Rz:=15), v200, z200, Tooldata_9;
MoveJ RelTool (starting_position, -75,60, -612.1 \Rx:=1.9, \Ry:=-15, \Rz:=15), v200, z200, Tooldata_9;
MoveJ RelTool (starting_position, -79,60, -610.3 \Rx:=1.9, \Ry:=-15.3, \Rz:=15), v200, z200, Tooldata_9;
MoveJ RelTool (starting_position, -83,60, -607.4 \Rx:=1.9, \Ry:=-15.9, \Rz:=15), v200, z200, Tooldata_9;
MoveJ RelTool (starting_position, -86,60, -603.6 \Rx:=1.9, \Ry:=-16.2, \Rz:=15), v200, z200, Tooldata_9;
MoveJ RelTool (starting_position, -88,60, -598.7 \Rx:=1.8, \Ry:=-16.5, \Rz:=15), v200, z200, Tooldata_9;
MoveJ RelTool (starting_position, -90,60, -593.1 \Rx:=1.8, \Ry:=-16.5, \Rz:=15), v200, z200, Tooldata_9;
MoveJ RelTool (starting_position, -91,60, -586.7 \Rx:=1.8, \Ry:=-16.5, \Rz:=15), v200, z200, Tooldata_9;
MoveJ RelTool (starting_position, -91,60, -579.6 \Rx:=1.8, \Ry:=-16.5, \Rz:=15), v200, z200, Tooldata_9;
MoveJ RelTool (starting_position, -90,60, -571.7 \Rx:=1.7, \Ry:=-16.5, \Rz:=15), v200, z200, Tooldata_9;
MoveJ RelTool (starting_position, -88,60, -563.2 \Rx:=1.7, \Ry:=-16.5, \Rz:=15), v200, z200, Tooldata_9;
MoveJ RelTool (starting_position, -86,60, -554.3 \Rx:=1.7, \Ry:=-16.2, \Rz:=15), v200, z200, Tooldata_9;
MoveJ RelTool (starting_position, -82,60, -544.9 \Rx:=1.7, \Ry:=-15.6, \Rz:=15), v200, z200, Tooldata_9;
MoveJ RelTool (starting_position, -78,60, -535.1 \Rx:=1.6, \Ry:=-15.3, \Rz:=15), v200, z200, Tooldata_9;
MoveJ RelTool (starting_position, -74,60, -524.8 \Rx:=1.6, \Ry:=-15, \Rz:=15), v200, z200, Tooldata_9;
MoveJ RelTool (starting_position, -68,60, -514.4 \Rx:=1.6, \Ry:=-14.4, \Rz:=15), v200, z200, Tooldata_9;
MoveJ RelTool (starting_position, -62,60, -504.4 \Rx:=1.5, \Ry:=-14.1, \Rz:=15), v200, z200, Tooldata_9;
MoveJ RelTool (starting_position, -55,60, -494.9 \Rx:=1.5, \Ry:=-13.5, \Rz:=15), v200, z200, Tooldata_9;
MoveJ RelTool (starting_position, -47,60, -486.3 \Rx:=1.5, \Ry:=-12.9, \Rz:=15), v200, z200, Tooldata_9;
MoveJ RelTool (starting_position, -39,60, -478.7 \Rx:=1.4, \Ry:=-12, \Rz:=15), v200, z200, Tooldata_9;
MoveJ RelTool (starting_position, -30,60, -472.3 \Rx:=1.4, \Ry:=-11.1, \Rz:=15), v200, z200, Tooldata_9;
MoveJ RelTool (starting_position, -21,60, -467 \Rx:=1.3, \Ry:=-9.9, \Rz:=15), v200, z200, Tooldata_9;
MoveJ RelTool (starting_position, -11,60, -462.9 \Rx:=1.3, \Ry:=-9, \Rz:=15), v200, z200, Tooldata_9;
MoveJ RelTool (starting_position, -2,60, -459.9 \Rx:=1.3, \Ry:=-8.1, \Rz:=15), v200, z200, Tooldata_9;
MoveJ RelTool (starting_position, 8,60, -457.7 \Rx:=1.2, \Ry:=-7.5, \Rz:=15), v200, z200, Tooldata_9;
MoveJ RelTool (starting_position, 17,60, -456.4 \Rx:=1.2, \Ry:=-6.9, \Rz:=15), v200, z200, Tooldata_9;
MoveJ RelTool (starting_position, 27,60, -456.1 \Rx:=1.1, \Ry:=-5.7, \Rz:=15), v200, z200, Tooldata_9;
MoveJ RelTool (starting_position, 36,60, -456.6 \Rx:=1, \Ry:=-4.8, \Rz:=15), v200, z200, Tooldata_9;
MoveJ RelTool (starting_position, 45,60, -458 \Rx:=1, \Ry:=-3.9, \Rz:=15), v200, z200, Tooldata_9;
MoveJ RelTool (starting_position, 53,60, -460.3 \Rx:=0.9, \Ry:=-3.3, \Rz:=15), v200, z200, Tooldata_9;
MoveJ RelTool (starting_position, 62,60, -463.4 \Rx:=0.9, \Ry:=-2.4, \Rz:=15), v200, z200, Tooldata_9;
MoveJ RelTool (starting_position, 69,60, -467.1 \Rx:=0.9, \Ry:=-1.8, \Rz:=15), v200, z200, Tooldata_9;
MoveJ RelTool (starting_position, 76,60, -471.5 \Rx:=0.8, \Ry:=-1.2, \Rz:=15), v200, z200, Tooldata_9;
MoveJ RelTool (starting_position, 82,60, -476.5 \Rx:=0.7, \Ry:=-0.6, \Rz:=15), v200, z200, Tooldata_9;
MoveJ RelTool (starting_position, 88,60, -481.8 \Rx:=0.7, \Ry:=-0, \Rz:=15), v200, z200, Tooldata_9;
MoveJ RelTool (starting_position, 93,60, -487.3 \Rx:=0.6, \Ry:=0.3, \Rz:=15), v200, z200, Tooldata_9;
MoveJ RelTool (starting_position, 97,60, -492.9 \Rx:=0.6, \Ry:=0.6, \Rz:=15), v200, z200, Tooldata_9;
MoveJ RelTool (starting_position, 101,60, -498.4 \Rx:=0.5, \Ry:=0.9, \Rz:=15), v200, z200, Tooldata_9;
MoveJ RelTool (starting_position, 104,60, -503.8 \Rx:=0.5, \Ry:=1.2, \Rz:=15), v200, z200, Tooldata_9;
MoveJ RelTool (starting_position, 106,60, -508.8 \Rx:=0.5, \Ry:=1.5, \Rz:=15), v200, z200, Tooldata_9;
MoveJ RelTool (starting_position, 108,60, -513.5 \Rx:=0.4, \Ry:=1.5, \Rz:=15), v200, z200, Tooldata_9;
MoveJ RelTool (starting_position, 109,60, -517.6 \Rx:=0.4, \Ry:=1.5, \Rz:=15), v200, z200, Tooldata_9;
MoveJ RelTool (starting_position, 110,60, -521.1 \Rx:=0.3, \Ry:=1.5, \Rz:=15), v200, z200, Tooldata_9;
MoveJ RelTool (starting_position, 110,60, -523.9 \Rx:=0.3, \Ry:=1.5, \Rz:=15), v200, z200, Tooldata_9;
MoveJ RelTool (starting_position, 110,60, -525.9 \Rx:=0.2, \Ry:=1.5, \Rz:=15), v200, z200, Tooldata_9;
MoveJ RelTool (starting_position, 110,60, -527 \Rx:=0.1, \Ry:=1.5, \Rz:=15), v200, z200, Tooldata_9;
MoveJ RelTool (starting_position, 109,60, -527.2 \Rx:=0.1, \Ry:=1.2, \Rz:=15), v200, z200, Tooldata_9;
MoveJ RelTool (starting_position, 109,60, -526.3 \Rx:=0, \Ry:=1.2, \Rz:=15), v200, z200, Tooldata_9;
MoveJ RelTool (starting_position, 108,60, -524.3 \Rx:=-0, \Ry:=1.2, \Rz:=15), v200, z200, Tooldata_9;
MoveJ RelTool (starting_position, 108,60, -521 \Rx:=-0.1, \Ry:=1.2, \Rz:=15), v200, z200, Tooldata_9;
MoveJ RelTool (starting_position, 107,60, -516.3 \Rx:=-0.2, \Ry:=0.9, \Rz:=15), v200, z200, Tooldata_9;
MoveJ RelTool (starting_position, 107,60, -510.5 \Rx:=-0.2, \Ry:=0.9, \Rz:=15), v200, z200, Tooldata_9;
MoveJ RelTool (starting_position, 106,60, -503.9 \Rx:=-0.3, \Ry:=0.9, \Rz:=15), v200, z200, Tooldata_9;
MoveJ RelTool (starting_position, 106,60, -497.1 \Rx:=-0.4, \Ry:=0.9, \Rz:=15), v200, z200, Tooldata_9;
MoveJ RelTool (starting_position, 106,60, -490 \Rx:=-0.4, \Ry:=0.6, \Rz:=15), v200, z200, Tooldata_9;
MoveJ RelTool (starting_position, 106,60, -483.3 \Rx:=-0.5, \Ry:=0.9, \Rz:=15), v200, z200, Tooldata_9;
MoveJ RelTool (starting_position, 107,60, -477.5 \Rx:=-0.6, \Ry:=0.9, \Rz:=15), v200, z200, Tooldata_9;
MoveJ RelTool (starting_position, 107,60, -473.1 \Rx:=-0.7, \Ry:=0.9, \Rz:=15), v200, z200, Tooldata_9;
MoveJ RelTool (starting_position, 108,60, -470.4 \Rx:=-0.7, \Ry:=1.2, \Rz:=15), v200, z200, Tooldata_9;
MoveJ RelTool (starting_position, 110,60, -469.1 \Rx:=-0.8, \Ry:=1.2, \Rz:=15), v200, z200, Tooldata_9;
MoveJ RelTool (starting_position, 111,60, -468.9 \Rx:=-0.9, \Ry:=1.2, \Rz:=15), v200, z200, Tooldata_9;
MoveJ RelTool (starting_position, 113,60, -469.2 \Rx:=-0.9, \Ry:=1.2, \Rz:=15), v200, z200, Tooldata_9;
MoveJ RelTool (starting_position, 115,60, -469.6 \Rx:=-1, \Ry:=1.5, \Rz:=15), v200, z200, Tooldata_9;
MoveJ RelTool (starting_position, 117,60, -469.8 \Rx:=-1.1, \Ry:=2.1, \Rz:=15), v200, z200, Tooldata_9;
MoveJ RelTool (starting_position, 119,56, -469.8 \Rx:=-1.2, \Ry:=2.1, \Rz:=14), v200, z200, Tooldata_9;
MoveJ RelTool (starting_position, 121,56, -469.7 \Rx:=-1.2, \Ry:=2.1, \Rz:=14), v200, z200, Tooldata_9;
MoveJ RelTool (starting_position, 124,56, -469.8 \Rx:=-1.3, \Ry:=2.4, \Rz:=14), v200, z200, Tooldata_9;
MoveJ RelTool (starting_position, 126,56, -470.3 \Rx:=-1.4, \Ry:=2.7, \Rz:=14), v200, z200, Tooldata_9;
MoveJ RelTool (starting_position, 129,56, -471.4 \Rx:=-1.4, \Ry:=3, \Rz:=14), v200, z200, Tooldata_9;
MoveJ RelTool (starting_position, 131,56, -473.1 \Rx:=-1.5, \Ry:=3.3, \Rz:=14), v200, z200, Tooldata_9;
MoveJ RelTool (starting_position, 134,56, -475.3 \Rx:=-1.6, \Ry:=3.6, \Rz:=14), v200, z200, Tooldata_9;
MoveJ RelTool (starting_position, 136,56, -477.8 \Rx:=-1.7, \Ry:=3.6, \Rz:=14), v200, z200, Tooldata_9;
MoveJ RelTool (starting_position, 138,56, -480.6 \Rx:=-1.7, \Ry:=3.9, \Rz:=14), v200, z200, Tooldata_9;
MoveJ RelTool (starting_position, 140,56, -483.4 \Rx:=-1.8, \Ry:=4.2, \Rz:=14), v200, z200, Tooldata_9;
MoveJ RelTool (starting_position, 142,56, -486.5 \Rx:=-1.9, \Ry:=4.2, \Rz:=14), v200, z200, Tooldata_9;
MoveJ RelTool (starting_position, 144,56, -489.6 \Rx:=-1.9, \Ry:=4.5, \Rz:=14), v200, z200, Tooldata_9;
MoveJ RelTool (starting_position, 145,56, -492.4 \Rx:=-2, \Ry:=4.5, \Rz:=14), v200, z200, Tooldata_9;
MoveJ RelTool (starting_position, 146,56, -494.9 \Rx:=-2, \Ry:=4.8, \Rz:=14), v200, z200, Tooldata_9;
MoveJ RelTool (starting_position, 147,56, -497.1 \Rx:=-2.1, \Ry:=4.5, \Rz:=14), v200, z200, Tooldata_9;
MoveJ RelTool (starting_position, 148,56, -498.9 \Rx:=-2.2, \Ry:=4.5, \Rz:=14), v200, z200, Tooldata_9;
MoveJ RelTool (starting_position, 149,56, -500.5 \Rx:=-2.3, \Ry:=4.8, \Rz:=14), v200, z200, Tooldata_9;
MoveJ RelTool (starting_position, 149,56, -501.7 \Rx:=-2.3, \Ry:=4.8, \Rz:=14), v200, z200, Tooldata_9;
MoveJ RelTool (starting_position, 149,56, -502.6 \Rx:=-2.4, \Ry:=4.8, \Rz:=14), v200, z200, Tooldata_9;
MoveJ RelTool (starting_position, 150,56, -503.2 \Rx:=-2.4, \Ry:=4.8, \Rz:=14), v200, z200, Tooldata_9;
MoveJ RelTool (starting_position, 150,56, -503.6 \Rx:=-2.5, \Ry:=4.8, \Rz:=14), v200, z200, Tooldata_9;
MoveJ RelTool (starting_position, 150,56, -503.8 \Rx:=-2.5, \Ry:=4.8, \Rz:=14), v200, z200, Tooldata_9;
MoveJ RelTool (starting_position, 150,56, -503.9 \Rx:=-2.6, \Ry:=4.8, \Rz:=14), v200, z200, Tooldata_9;
MoveJ RelTool (starting_position, 150,56, -503.9 \Rx:=-2.6, \Ry:=4.8, \Rz:=14), v200, z200, Tooldata_9;
MoveJ RelTool (starting_position, 150,56, -503.8 \Rx:=-2.6, \Ry:=4.8, \Rz:=14), v200, z200, Tooldata_9;
MoveJ RelTool (starting_position, 151,56, -503.7 \Rx:=-2.7, \Ry:=4.8, \Rz:=14), v200, z200, Tooldata_9;
MoveJ RelTool (starting_position, 151,56, -503.5 \Rx:=-2.7, \Ry:=4.8, \Rz:=14), v200, z200, Tooldata_9;
MoveJ RelTool (starting_position, 151,56, -503.2 \Rx:=-2.7, \Ry:=4.8, \Rz:=14), v200, z200, Tooldata_9;
MoveJ RelTool (starting_position, 152,56, -502.7 \Rx:=-2.8, \Ry:=4.8, \Rz:=14), v200, z200, Tooldata_9;
MoveJ RelTool (starting_position, 152,56, -502.1 \Rx:=-2.8, \Ry:=4.8, \Rz:=14), v200, z200, Tooldata_9;
MoveJ RelTool (starting_position, 153,56, -501.6 \Rx:=-2.8, \Ry:=5.1, \Rz:=14), v200, z200, Tooldata_9;
MoveJ RelTool (starting_position, 154,56, -501 \Rx:=-2.9, \Ry:=5.1, \Rz:=14), v200, z200, Tooldata_9;
MoveJ RelTool (starting_position, 154,56, -500.5 \Rx:=-2.9, \Ry:=5.1, \Rz:=14), v200, z200, Tooldata_9;
MoveJ RelTool (starting_position, 155,56, -499.9 \Rx:=-2.9, \Ry:=5.4, \Rz:=14), v200, z200, Tooldata_9;
MoveJ RelTool (starting_position, 156,56, -499.5 \Rx:=-2.9, \Ry:=5.4, \Rz:=14), v200, z200, Tooldata_9;
MoveJ RelTool (starting_position, 156,56, -499.1 \Rx:=-2.9, \Ry:=5.4, \Rz:=14), v200, z200, Tooldata_9;
MoveJ RelTool (starting_position, 157,56, -498.9 \Rx:=-2.9, \Ry:=5.4, \Rz:=14), v200, z200, Tooldata_9;
MoveJ RelTool (starting_position, 158,56, -499 \Rx:=-2.9, \Ry:=5.4, \Rz:=14), v200, z200, Tooldata_9;
MoveJ RelTool (starting_position, 159,52, -499.3 \Rx:=-2.9, \Ry:=5.1, \Rz:=13), v200, z200, Tooldata_9;
MoveJ RelTool (starting_position, 160,52, -499.9 \Rx:=-2.8, \Ry:=5.4, \Rz:=13), v200, z200, Tooldata_9;
MoveJ RelTool (starting_position, 161,52, -500.7 \Rx:=-2.8, \Ry:=5.7, \Rz:=13), v200, z200, Tooldata_9;
MoveJ RelTool (starting_position, 162,52, -501.8 \Rx:=-2.7, \Ry:=6, \Rz:=13), v200, z200, Tooldata_9;
MoveJ RelTool (starting_position, 163,52, -503.2 \Rx:=-2.7, \Ry:=6, \Rz:=13), v200, z200, Tooldata_9;
MoveJ RelTool (starting_position, 164,52, -504.9 \Rx:=-2.6, \Ry:=6, \Rz:=13), v200, z200, Tooldata_9;
MoveJ RelTool (starting_position, 165,52, -506.9 \Rx:=-2.6, \Ry:=6, \Rz:=13), v200, z200, Tooldata_9;
MoveJ RelTool (starting_position, 166,52, -509 \Rx:=-2.5, \Ry:=6.3, \Rz:=13), v200, z200, Tooldata_9;
MoveJ RelTool (starting_position, 167,52, -511.1 \Rx:=-2.4, \Ry:=6.3, \Rz:=13), v200, z200, Tooldata_9;
MoveJ RelTool (starting_position, 168,52, -513.3 \Rx:=-2.4, \Ry:=6.6, \Rz:=13), v200, z200, Tooldata_9;
MoveJ RelTool (starting_position, 169,52, -515.4 \Rx:=-2.3, \Ry:=6.6, \Rz:=13), v200, z200, Tooldata_9;
MoveJ RelTool (starting_position, 169,52, -517.2 \Rx:=-2.2, \Ry:=6.6, \Rz:=13), v200, z200, Tooldata_9;
MoveJ RelTool (starting_position, 170,52, -518.8 \Rx:=-2.1, \Ry:=6.6, \Rz:=13), v200, z200, Tooldata_9;
MoveJ RelTool (starting_position, 170,52, -520 \Rx:=-2, \Ry:=6.6, \Rz:=13), v200, z200, Tooldata_9;
MoveJ RelTool (starting_position, 169,52, -521.1 \Rx:=-1.8, \Ry:=6.6, \Rz:=13), v200, z200, Tooldata_9;
MoveJ RelTool (starting_position, 169,52, -522 \Rx:=-1.7, \Ry:=6.6, \Rz:=13), v200, z200, Tooldata_9;
MoveJ RelTool (starting_position, 168,52, -522.8 \Rx:=-1.6, \Ry:=6.6, \Rz:=13), v200, z200, Tooldata_9;
MoveJ RelTool (starting_position, 168,52, -523.7 \Rx:=-1.5, \Ry:=6.3, \Rz:=13), v200, z200, Tooldata_9;
MoveJ RelTool (starting_position, 166,52, -524.8 \Rx:=-1.4, \Ry:=6.3, \Rz:=13), v200, z200, Tooldata_9;
MoveJ RelTool (starting_position, 165,52, -526 \Rx:=-1.2, \Ry:=6.3, \Rz:=13), v200, z200, Tooldata_9;
MoveJ RelTool (starting_position, 164,52, -527.5 \Rx:=-1.1, \Ry:=6, \Rz:=13), v200, z200, Tooldata_9;
MoveJ RelTool (starting_position, 162,52, -529.1 \Rx:=-1, \Ry:=6, \Rz:=13), v200, z200, Tooldata_9;
MoveJ RelTool (starting_position, 160,52, -530.9 \Rx:=-0.8, \Ry:=5.7, \Rz:=13), v200, z200, Tooldata_9;
MoveJ RelTool (starting_position, 157,52, -532.7 \Rx:=-0.7, \Ry:=5.7, \Rz:=13), v200, z200, Tooldata_9;
MoveJ RelTool (starting_position, 155,52, -534.8 \Rx:=-0.5, \Ry:=5.4, \Rz:=13), v200, z200, Tooldata_9;
MoveJ RelTool (starting_position, 152,52, -536.9 \Rx:=-0.4, \Ry:=5.1, \Rz:=13), v200, z200, Tooldata_9;
MoveJ RelTool (starting_position, 149,52, -539.2 \Rx:=-0.3, \Ry:=4.8, \Rz:=13), v200, z200, Tooldata_9;
MoveJ RelTool (starting_position, 146,48, -541.5 \Rx:=-0.1, \Ry:=4.5, \Rz:=12), v200, z200, Tooldata_9;
MoveJ RelTool (starting_position, 142,48, -543.8 \Rx:=0, \Ry:=4.2, \Rz:=12), v200, z200, Tooldata_9;
MoveJ RelTool (starting_position, 139,48, -545.9 \Rx:=0.2, \Ry:=3.9, \Rz:=12), v200, z200, Tooldata_9;
MoveJ RelTool (starting_position, 135,48, -547.7 \Rx:=0.3, \Ry:=3.6, \Rz:=12), v200, z200, Tooldata_9;
MoveJ RelTool (starting_position, 131,48, -549.1 \Rx:=0.4, \Ry:=3.3, \Rz:=12), v200, z200, Tooldata_9;
MoveJ RelTool (starting_position, 128,48, -550.2 \Rx:=0.6, \Ry:=2.7, \Rz:=12), v200, z200, Tooldata_9;
MoveJ RelTool (starting_position, 124,48, -550.9 \Rx:=0.7, \Ry:=2.4, \Rz:=12), v200, z200, Tooldata_9;
MoveJ RelTool (starting_position, 120,48, -551.2 \Rx:=0.9, \Ry:=2.1, \Rz:=12), v200, z200, Tooldata_9;
MoveJ RelTool (starting_position, 116,48, -551.3 \Rx:=1, \Ry:=1.8, \Rz:=12), v200, z200, Tooldata_9;
MoveJ RelTool (starting_position, 113,48, -551.1 \Rx:=1.2, \Ry:=1.5, \Rz:=12), v200, z200, Tooldata_9;
MoveJ RelTool (starting_position, 109,48, -550.7 \Rx:=1.3, \Ry:=1.2, \Rz:=12), v200, z200, Tooldata_9;
MoveJ RelTool (starting_position, 106,48, -550 \Rx:=1.5, \Ry:=0.9, \Rz:=12), v200, z200, Tooldata_9;
MoveJ RelTool (starting_position, 103,48, -549.2 \Rx:=1.6, \Ry:=0.6, \Rz:=12), v200, z200, Tooldata_9;
MoveJ RelTool (starting_position, 100,48, -548.3 \Rx:=1.8, \Ry:=0.3, \Rz:=12), v200, z200, Tooldata_9;
MoveJ RelTool (starting_position, 97,48, -547.4 \Rx:=1.9, \Ry:=-0, \Rz:=12), v200, z200, Tooldata_9;
MoveJ RelTool (starting_position, 95,48, -546.4 \Rx:=2, \Ry:=-0.3, \Rz:=12), v200, z200, Tooldata_9;
MoveJ RelTool (starting_position, 93,48, -545.3 \Rx:=2.1, \Ry:=-0.3, \Rz:=12), v200, z200, Tooldata_9;
MoveJ RelTool (starting_position, 91,48, -544 \Rx:=2.2, \Ry:=-0.6, \Rz:=12), v200, z200, Tooldata_9;
MoveJ RelTool (starting_position, 89,48, -542.6 \Rx:=2.3, \Ry:=-0.6, \Rz:=12), v200, z200, Tooldata_9;
MoveJ RelTool (starting_position, 88,48, -540.9 \Rx:=2.4, \Ry:=-0.9, \Rz:=12), v200, z200, Tooldata_9;
MoveJ RelTool (starting_position, 87,48, -538.9 \Rx:=2.5, \Ry:=-0.9, \Rz:=12), v200, z200, Tooldata_9;
MoveJ RelTool (starting_position, 86,48, -536.8 \Rx:=2.6, \Ry:=-0.9, \Rz:=12), v200, z200, Tooldata_9;
MoveJ RelTool (starting_position, 86,48, -534.6 \Rx:=2.7, \Ry:=-0.9, \Rz:=12), v200, z200, Tooldata_9;
MoveJ RelTool (starting_position, 86,44, -532.3 \Rx:=2.8, \Ry:=-0.9, \Rz:=11), v200, z200, Tooldata_9;
MoveJ RelTool (starting_position, 86,44, -530.3 \Rx:=2.9, \Ry:=-0.9, \Rz:=11), v200, z200, Tooldata_9;
MoveJ RelTool (starting_position, 87,44, -528.5 \Rx:=2.9, \Ry:=-0.9, \Rz:=11), v200, z200, Tooldata_9;
MoveJ RelTool (starting_position, 88,44, -527.1 \Rx:=3, \Ry:=-0.9, \Rz:=11), v200, z200, Tooldata_9;
MoveJ RelTool (starting_position, 89,44, -526.2 \Rx:=3, \Ry:=-0.6, \Rz:=11), v200, z200, Tooldata_9;
MoveJ RelTool (starting_position, 90,44, -525.7 \Rx:=3.1, \Ry:=-0.6, \Rz:=11), v200, z200, Tooldata_9;
MoveJ RelTool (starting_position, 92,44, -525.7 \Rx:=3.1, \Ry:=-0.3, \Rz:=11), v200, z200, Tooldata_9;
MoveJ RelTool (starting_position, 94,44, -526.3 \Rx:=3.2, \Ry:=-0, \Rz:=11), v200, z200, Tooldata_9;
MoveJ RelTool (starting_position, 96,44, -527.3 \Rx:=3.2, \Ry:=0, \Rz:=11), v200, z200, Tooldata_9;
MoveJ RelTool (starting_position, 98,44, -528.6 \Rx:=3.2, \Ry:=0.3, \Rz:=11), v200, z200, Tooldata_9;
MoveJ RelTool (starting_position, 100,44, -530.1 \Rx:=3.2, \Ry:=0.3, \Rz:=11), v200, z200, Tooldata_9;
MoveJ RelTool (starting_position, 103,44, -531.5 \Rx:=3.2, \Ry:=0.6, \Rz:=11), v200, z200, Tooldata_9;
MoveJ RelTool (starting_position, 105,44, -532.7 \Rx:=3.2, \Ry:=0.9, \Rz:=11), v200, z200, Tooldata_9;
MoveJ RelTool (starting_position, 107,44, -533.8 \Rx:=3.2, \Ry:=1.2, \Rz:=11), v200, z200, Tooldata_9;
MoveJ RelTool (starting_position, 110,44, -534.5 \Rx:=3.2, \Ry:=1.2, \Rz:=11), v200, z200, Tooldata_9;
MoveJ RelTool (starting_position, 112,44, -534.9 \Rx:=3.2, \Ry:=1.5, \Rz:=11), v200, z200, Tooldata_9;
MoveJ RelTool (starting_position, 115,44, -534.9 \Rx:=3.2, \Ry:=1.8, \Rz:=11), v200, z200, Tooldata_9;
MoveJ RelTool (starting_position, 117,44, -534.6 \Rx:=3.2, \Ry:=2.1, \Rz:=11), v200, z200, Tooldata_9;
MoveJ RelTool (starting_position, 119,44, -534.3 \Rx:=3.2, \Ry:=2.1, \Rz:=11), v200, z200, Tooldata_9;
MoveJ RelTool (starting_position, 122,40, -533.9 \Rx:=3.1, \Ry:=2.4, \Rz:=10), v200, z200, Tooldata_9;
MoveJ RelTool (starting_position, 124,40, -533.7 \Rx:=3.1, \Ry:=2.7, \Rz:=10), v200, z200, Tooldata_9;
MoveJ RelTool (starting_position, 125,40, -533.6 \Rx:=3.1, \Ry:=2.7, \Rz:=10), v200, z200, Tooldata_9;
MoveJ RelTool (starting_position, 127,40, -533.8 \Rx:=3.1, \Ry:=3, \Rz:=10), v200, z200, Tooldata_9;
MoveJ RelTool (starting_position, 129,40, -534.2 \Rx:=3.1, \Ry:=3, \Rz:=10), v200, z200, Tooldata_9;
MoveJ RelTool (starting_position, 130,40, -534.8 \Rx:=3, \Ry:=3.3, \Rz:=10), v200, z200, Tooldata_9;
MoveJ RelTool (starting_position, 131,40, -535.7 \Rx:=3, \Ry:=3.3, \Rz:=10), v200, z200, Tooldata_9;
MoveJ RelTool (starting_position, 132,40, -536.7 \Rx:=2.9, \Ry:=3.3, \Rz:=10), v200, z200, Tooldata_9;
MoveJ RelTool (starting_position, 133,40, -537.8 \Rx:=2.9, \Ry:=3.3, \Rz:=10), v200, z200, Tooldata_9;
MoveJ RelTool (starting_position, 134,40, -539.1 \Rx:=2.9, \Ry:=3.6, \Rz:=10), v200, z200, Tooldata_9;
MoveJ RelTool (starting_position, 134,40, -540.5 \Rx:=2.8, \Ry:=3.6, \Rz:=10), v200, z200, Tooldata_9;
MoveJ RelTool (starting_position, 134,40, -542.1 \Rx:=2.8, \Ry:=3.6, \Rz:=10), v200, z200, Tooldata_9;
MoveJ RelTool (starting_position, 133,40, -543.8 \Rx:=2.8, \Ry:=3.6, \Rz:=10), v200, z200, Tooldata_9;
MoveJ RelTool (starting_position, 133,40, -545.5 \Rx:=2.7, \Ry:=3.6, \Rz:=10), v200, z200, Tooldata_9;
MoveJ RelTool (starting_position, 132,40, -547.3 \Rx:=2.7, \Ry:=3.3, \Rz:=10), v200, z200, Tooldata_9;
MoveJ RelTool (starting_position, 131,40, -549.1 \Rx:=2.6, \Ry:=3.3, \Rz:=10), v200, z200, Tooldata_9;
MoveJ RelTool (starting_position, 129,40, -550.9 \Rx:=2.6, \Ry:=3, \Rz:=10), v200, z200, Tooldata_9;
MoveJ RelTool (starting_position, 127,40, -552.5 \Rx:=2.6, \Ry:=3, \Rz:=10), v200, z200, Tooldata_9;
MoveJ RelTool (starting_position, 126,36, -553.9 \Rx:=2.5, \Ry:=2.7, \Rz:=9), v200, z200, Tooldata_9;
MoveJ RelTool (starting_position, 123,36, -555 \Rx:=2.5, \Ry:=2.7, \Rz:=9), v200, z200, Tooldata_9;
MoveJ RelTool (starting_position, 121,36, -555.9 \Rx:=2.4, \Ry:=2.4, \Rz:=9), v200, z200, Tooldata_9;
MoveJ RelTool (starting_position, 118,36, -556.5 \Rx:=2.4, \Ry:=2.1, \Rz:=9), v200, z200, Tooldata_9;
MoveJ RelTool (starting_position, 116,36, -556.9 \Rx:=2.4, \Ry:=1.8, \Rz:=9), v200, z200, Tooldata_9;
MoveJ RelTool (starting_position, 113,36, -557.2 \Rx:=2.3, \Ry:=1.8, \Rz:=9), v200, z200, Tooldata_9;
MoveJ RelTool (starting_position, 109,36, -557.4 \Rx:=2.3, \Ry:=1.5, \Rz:=9), v200, z200, Tooldata_9;
MoveJ RelTool (starting_position, 106,36, -557.5 \Rx:=2.3, \Ry:=1.2, \Rz:=9), v200, z200, Tooldata_9;
MoveJ RelTool (starting_position, 103,36, -557.5 \Rx:=2.2, \Ry:=0.6, \Rz:=9), v200, z200, Tooldata_9;
MoveJ RelTool (starting_position, 99,36, -557.5 \Rx:=2.2, \Ry:=0.3, \Rz:=9), v200, z200, Tooldata_9;
MoveJ RelTool (starting_position, 95,36, -557.5 \Rx:=2.2, \Ry:=0, \Rz:=9), v200, z200, Tooldata_9;
MoveJ RelTool (starting_position, 91,36, -557.5 \Rx:=2.2, \Ry:=-0.3, \Rz:=9), v200, z200, Tooldata_9;
MoveJ RelTool (starting_position, 88,36, -557.5 \Rx:=2.2, \Ry:=-0.6, \Rz:=9), v200, z200, Tooldata_9;
MoveJ RelTool (starting_position, 84,36, -557.5 \Rx:=2.2, \Ry:=-0.9, \Rz:=9), v200, z200, Tooldata_9;
MoveJ RelTool (starting_position, 80,36, -557.5 \Rx:=2.2, \Ry:=-1.2, \Rz:=9), v200, z200, Tooldata_9;
MoveJ RelTool (starting_position, 76,36, -557.5 \Rx:=2.2, \Ry:=-1.5, \Rz:=9), v200, z200, Tooldata_9;
MoveJ RelTool (starting_position, 72,36, -557.5 \Rx:=2.1, \Ry:=-2.1, \Rz:=9), v200, z200, Tooldata_9;
MoveJ RelTool (starting_position, 69,32, -557.3 \Rx:=2.1, \Ry:=-2.4, \Rz:=8), v200, z200, Tooldata_9;
MoveJ RelTool (starting_position, 65,32, -557 \Rx:=2.1, \Ry:=-2.7, \Rz:=8), v200, z200, Tooldata_9;
MoveJ RelTool (starting_position, 61,32, -556.6 \Rx:=2.1, \Ry:=-3, \Rz:=8), v200, z200, Tooldata_9;
MoveJ RelTool (starting_position, 58,32, -555.9 \Rx:=2.1, \Ry:=-3.3, \Rz:=8), v200, z200, Tooldata_9;
MoveJ RelTool (starting_position, 55,32, -555.1 \Rx:=2.1, \Ry:=-3.6, \Rz:=8), v200, z200, Tooldata_9;
MoveJ RelTool (starting_position, 51,32, -554 \Rx:=2.1, \Ry:=-3.9, \Rz:=8), v200, z200, Tooldata_9;
MoveJ RelTool (starting_position, 48,32, -552.6 \Rx:=2.1, \Ry:=-3.9, \Rz:=8), v200, z200, Tooldata_9;
MoveJ RelTool (starting_position, 45,32, -551.1 \Rx:=2.2, \Ry:=-4.2, \Rz:=8), v200, z200, Tooldata_9;
MoveJ RelTool (starting_position, 42,32, -549.4 \Rx:=2.2, \Ry:=-4.8, \Rz:=8), v200, z200, Tooldata_9;
MoveJ RelTool (starting_position, 39,32, -547.8 \Rx:=2.2, \Ry:=-4.8, \Rz:=8), v200, z200, Tooldata_9;
MoveJ RelTool (starting_position, 36,32, -546.2 \Rx:=2.2, \Ry:=-5.1, \Rz:=8), v200, z200, Tooldata_9;
MoveJ RelTool (starting_position, 33,32, -544.8 \Rx:=2.2, \Ry:=-5.4, \Rz:=8), v200, z200, Tooldata_9;
MoveJ RelTool (starting_position, 30,32, -543.5 \Rx:=2.2, \Ry:=-5.7, \Rz:=8), v200, z200, Tooldata_9;
MoveJ RelTool (starting_position, 28,32, -542.3 \Rx:=2.3, \Ry:=-6, \Rz:=8), v200, z200, Tooldata_9;
MoveJ RelTool (starting_position, 25,32, -541.3 \Rx:=2.3, \Ry:=-6, \Rz:=8), v200, z200, Tooldata_9;
MoveJ RelTool (starting_position, 22,32, -540.3 \Rx:=2.3, \Ry:=-6.3, \Rz:=8), v200, z200, Tooldata_9;
MoveJ RelTool (starting_position, 20,28, -539.2 \Rx:=2.4, \Ry:=-6.6, \Rz:=7), v200, z200, Tooldata_9;
MoveJ RelTool (starting_position, 18,28, -538.1 \Rx:=2.4, \Ry:=-6.9, \Rz:=7), v200, z200, Tooldata_9;
MoveJ RelTool (starting_position, 16,28, -536.9 \Rx:=2.4, \Ry:=-6.9, \Rz:=7), v200, z200, Tooldata_9;
MoveJ RelTool (starting_position, 13,28, -535.5 \Rx:=2.5, \Ry:=-6.9, \Rz:=7), v200, z200, Tooldata_9;
MoveJ RelTool (starting_position, 11,28, -534.2 \Rx:=2.5, \Ry:=-7.2, \Rz:=7), v200, z200, Tooldata_9;
MoveJ RelTool (starting_position, 9,28, -532.8 \Rx:=2.5, \Ry:=-7.5, \Rz:=7), v200, z200, Tooldata_9;
MoveJ RelTool (starting_position, 8,28, -531.5 \Rx:=2.6, \Ry:=-7.5, \Rz:=7), v200, z200, Tooldata_9;
MoveJ RelTool (starting_position, 6,28, -530.4 \Rx:=2.7, \Ry:=-7.8, \Rz:=7), v200, z200, Tooldata_9;
MoveJ RelTool (starting_position, 4,28, -529.5 \Rx:=2.7, \Ry:=-8.1, \Rz:=7), v200, z200, Tooldata_9;
MoveJ RelTool (starting_position, 3,28, -528.7 \Rx:=2.7, \Ry:=-8.1, \Rz:=7), v200, z200, Tooldata_9;
MoveJ RelTool (starting_position, 1,28, -528.2 \Rx:=2.8, \Ry:=-8.1, \Rz:=7), v200, z200, Tooldata_9;
MoveJ RelTool (starting_position, 0,28, -527.8 \Rx:=2.8, \Ry:=-8.1, \Rz:=7), v200, z200, Tooldata_9;
MoveJ RelTool (starting_position, -2,28, -527.6 \Rx:=2.9, \Ry:=-8.4, \Rz:=7), v200, z200, Tooldata_9;
MoveJ RelTool (starting_position, -3,28, -527.4 \Rx:=2.9, \Ry:=-8.4, \Rz:=7), v200, z200, Tooldata_9;
MoveJ RelTool (starting_position, -4,28, -527.3 \Rx:=3, \Ry:=-8.7, \Rz:=7), v200, z200, Tooldata_9;
MoveJ RelTool (starting_position, -6,24, -527 \Rx:=3, \Ry:=-8.7, \Rz:=6), v200, z200, Tooldata_9;
MoveJ RelTool (starting_position, -7,24, -526.7 \Rx:=3.1, \Ry:=-8.7, \Rz:=6), v200, z200, Tooldata_9;
MoveJ RelTool (starting_position, -8,24, -526.2 \Rx:=3.1, \Ry:=-9, \Rz:=6), v200, z200, Tooldata_9;
MoveJ RelTool (starting_position, -10,24, -525.4 \Rx:=3.2, \Ry:=-9, \Rz:=6), v200, z200, Tooldata_9;
MoveJ RelTool (starting_position, -11,24, -524.3 \Rx:=3.2, \Ry:=-9.3, \Rz:=6), v200, z200, Tooldata_9;
MoveJ RelTool (starting_position, -12,24, -523 \Rx:=3.3, \Ry:=-9.3, \Rz:=6), v200, z200, Tooldata_9;
MoveJ RelTool (starting_position, -13,24, -521.4 \Rx:=3.3, \Ry:=-9.3, \Rz:=6), v200, z200, Tooldata_9;
MoveJ RelTool (starting_position, -14,24, -519.5 \Rx:=3.4, \Ry:=-9.6, \Rz:=6), v200, z200, Tooldata_9;
MoveJ RelTool (starting_position, -15,24, -517.5 \Rx:=3.4, \Ry:=-9.6, \Rz:=6), v200, z200, Tooldata_9;
MoveJ RelTool (starting_position, -16,24, -515.2 \Rx:=3.4, \Ry:=-9.6, \Rz:=6), v200, z200, Tooldata_9;
MoveJ RelTool (starting_position, -17,24, -513 \Rx:=3.5, \Ry:=-9.6, \Rz:=6), v200, z200, Tooldata_9;
MoveJ RelTool (starting_position, -18,24, -510.7 \Rx:=3.5, \Ry:=-9.9, \Rz:=6), v200, z200, Tooldata_9;
MoveJ RelTool (starting_position, -18,24, -508.4 \Rx:=3.5, \Ry:=-9.9, \Rz:=6), v200, z200, Tooldata_9;
MoveJ RelTool (starting_position, -19,24, -506 \Rx:=3.6, \Ry:=-9.9, \Rz:=6), v200, z200, Tooldata_9;
MoveJ RelTool (starting_position, -19,20, -503.5 \Rx:=3.6, \Ry:=-9.9, \Rz:=5), v200, z200, Tooldata_9;
MoveJ RelTool (starting_position, -19,20, -500.8 \Rx:=3.6, \Ry:=-9.9, \Rz:=5), v200, z200, Tooldata_9;
MoveJ RelTool (starting_position, -19,20, -498 \Rx:=3.7, \Ry:=-9.9, \Rz:=5), v200, z200, Tooldata_9;
MoveJ RelTool (starting_position, -20,20, -494.9 \Rx:=3.7, \Ry:=-9.9, \Rz:=5), v200, z200, Tooldata_9;
MoveJ RelTool (starting_position, -20,20, -491.7 \Rx:=3.7, \Ry:=-9.9, \Rz:=5), v200, z200, Tooldata_9;
MoveJ RelTool (starting_position, -20,20, -488.5 \Rx:=3.8, \Ry:=-9.9, \Rz:=5), v200, z200, Tooldata_9;
MoveJ RelTool (starting_position, -20,20, -485.4 \Rx:=3.8, \Ry:=-9.9, \Rz:=5), v200, z200, Tooldata_9;
MoveJ RelTool (starting_position, -20,20, -482.4 \Rx:=3.9, \Ry:=-9.9, \Rz:=5), v200, z200, Tooldata_9;
MoveJ RelTool (starting_position, -21,20, -479.5 \Rx:=3.9, \Ry:=-9.9, \Rz:=5), v200, z200, Tooldata_9;
MoveJ RelTool (starting_position, -21,20, -476.9 \Rx:=3.9, \Ry:=-9.9, \Rz:=5), v200, z200, Tooldata_9;
MoveJ RelTool (starting_position, -22,20, -474.7 \Rx:=3.9, \Ry:=-9.9, \Rz:=5), v200, z200, Tooldata_9;
MoveJ RelTool (starting_position, -23,20, -473.1 \Rx:=4, \Ry:=-9.9, \Rz:=5), v200, z200, Tooldata_9;
MoveJ RelTool (starting_position, -25,20, -471.9 \Rx:=4, \Ry:=-10.2, \Rz:=5), v200, z200, Tooldata_9;
MoveJ RelTool (starting_position, -27,20, -471.4 \Rx:=4, \Ry:=-10.2, \Rz:=5), v200, z200, Tooldata_9;
MoveJ RelTool (starting_position, -29,16, -471.3 \Rx:=4, \Ry:=-10.5, \Rz:=4), v200, z200, Tooldata_9;
MoveJ RelTool (starting_position, -31,16, -471.5 \Rx:=4, \Ry:=-10.8, \Rz:=4), v200, z200, Tooldata_9;
MoveJ RelTool (starting_position, -34,16, -472.2 \Rx:=4, \Ry:=-10.8, \Rz:=4), v200, z200, Tooldata_9;
MoveJ RelTool (starting_position, -37,16, -473.3 \Rx:=4.1, \Ry:=-11.1, \Rz:=4), v200, z200, Tooldata_9;
MoveJ RelTool (starting_position, -41,16, -474.6 \Rx:=4.1, \Ry:=-11.4, \Rz:=4), v200, z200, Tooldata_9;
MoveJ RelTool (starting_position, -45,16, -476 \Rx:=4.1, \Ry:=-12, \Rz:=4), v200, z200, Tooldata_9;
MoveJ RelTool (starting_position, -49,16, -477.5 \Rx:=4.1, \Ry:=-12.3, \Rz:=4), v200, z200, Tooldata_9;
MoveJ RelTool (starting_position, -54,16, -479 \Rx:=4.1, \Ry:=-12.6, \Rz:=4), v200, z200, Tooldata_9;
MoveJ RelTool (starting_position, -59,16, -480.1 \Rx:=4.1, \Ry:=-13.2, \Rz:=4), v200, z200, Tooldata_9;
MoveJ RelTool (starting_position, -64,16, -480.9 \Rx:=4.2, \Ry:=-13.5, \Rz:=4), v200, z200, Tooldata_9;
MoveJ RelTool (starting_position, -69,16, -481 \Rx:=4.2, \Ry:=-14.1, \Rz:=4), v200, z200, Tooldata_9;
MoveJ RelTool (starting_position, -75,16, -480.5 \Rx:=4.2, \Ry:=-14.7, \Rz:=4), v200, z200, Tooldata_9;
MoveJ RelTool (starting_position, -81,16, -479.2 \Rx:=4.2, \Ry:=-15, \Rz:=4), v200, z200, Tooldata_9;
MoveJ RelTool (starting_position, -87,16, -477.2 \Rx:=4.3, \Ry:=-15.6, \Rz:=4), v200, z200, Tooldata_9;
MoveJ RelTool (starting_position, -93,12, -474.6 \Rx:=4.3, \Ry:=-16.2, \Rz:=3), v200, z200, Tooldata_9;
MoveJ RelTool (starting_position, -99,12, -471.4 \Rx:=4.3, \Ry:=-16.8, \Rz:=3), v200, z200, Tooldata_9;
MoveJ RelTool (starting_position, -106,12, -467.9 \Rx:=4.3, \Ry:=-17.4, \Rz:=3), v200, z200, Tooldata_9;
MoveJ RelTool (starting_position, -112,12, -464.1 \Rx:=4.3, \Ry:=-18, \Rz:=3), v200, z200, Tooldata_9;
MoveJ RelTool (starting_position, -118,12, -460.1 \Rx:=4.3, \Ry:=-18.6, \Rz:=3), v200, z200, Tooldata_9;
MoveJ RelTool (starting_position, -124,12, -456 \Rx:=4.3, \Ry:=-18.9, \Rz:=3), v200, z200, Tooldata_9;
MoveJ RelTool (starting_position, -130,12, -452.1 \Rx:=4.3, \Ry:=-19.5, \Rz:=3), v200, z200, Tooldata_9;
MoveJ RelTool (starting_position, -136,12, -448.1 \Rx:=4.3, \Ry:=-20.1, \Rz:=3), v200, z200, Tooldata_9;
MoveJ RelTool (starting_position, -141,12, -444.1 \Rx:=4.3, \Ry:=-20.7, \Rz:=3), v200, z200, Tooldata_9;
MoveJ RelTool (starting_position, -147,12, -440.1 \Rx:=4.3, \Ry:=-21, \Rz:=3), v200, z200, Tooldata_9;
MoveJ RelTool (starting_position, -152,12, -436 \Rx:=4.3, \Ry:=-21.6, \Rz:=3), v200, z200, Tooldata_9;
MoveJ RelTool (starting_position, -156,12, -432 \Rx:=4.3, \Ry:=-21.9, \Rz:=3), v200, z200, Tooldata_9;
MoveJ RelTool (starting_position, -161,12, -427.9 \Rx:=4.3, \Ry:=-22.5, \Rz:=3), v200, z200, Tooldata_9;
MoveJ RelTool (starting_position, -164,12, -424 \Rx:=4.3, \Ry:=-22.8, \Rz:=3), v200, z200, Tooldata_9;
MoveJ RelTool (starting_position, -168,8, -420.1 \Rx:=4.3, \Ry:=-23.1, \Rz:=2), v200, z200, Tooldata_9;
MoveJ RelTool (starting_position, -170,8, -416.4 \Rx:=4.3, \Ry:=-23.4, \Rz:=2), v200, z200, Tooldata_9;
MoveJ RelTool (starting_position, -172,8, -412.7 \Rx:=4.3, \Ry:=-23.4, \Rz:=2), v200, z200, Tooldata_9;
MoveJ RelTool (starting_position, -174,8, -409.2 \Rx:=4.3, \Ry:=-23.7, \Rz:=2), v200, z200, Tooldata_9;
MoveJ RelTool (starting_position, -175,8, -405.6 \Rx:=4.3, \Ry:=-23.7, \Rz:=2), v200, z200, Tooldata_9;
MoveJ RelTool (starting_position, -175,8, -402.1 \Rx:=4.3, \Ry:=-23.7, \Rz:=2), v200, z200, Tooldata_9;
MoveJ RelTool (starting_position, -175,8, -398.4 \Rx:=4.3, \Ry:=-23.7, \Rz:=2), v200, z200, Tooldata_9;
MoveJ RelTool (starting_position, -174,8, -394.3 \Rx:=4.2, \Ry:=-23.7, \Rz:=2), v200, z200, Tooldata_9;
MoveJ RelTool (starting_position, -172,8, -389.9 \Rx:=4.2, \Ry:=-23.4, \Rz:=2), v200, z200, Tooldata_9;
MoveJ RelTool (starting_position, -170,8, -384.9 \Rx:=4.2, \Ry:=-23.4, \Rz:=2), v200, z200, Tooldata_9;
MoveJ RelTool (starting_position, -167,8, -379.3 \Rx:=4.2, \Ry:=-22.8, \Rz:=2), v200, z200, Tooldata_9;
MoveJ RelTool (starting_position, -164,8, -373.1 \Rx:=4.2, \Ry:=-22.8, \Rz:=2), v200, z200, Tooldata_9;
MoveJ RelTool (starting_position, -160,8, -366.4 \Rx:=4.2, \Ry:=-22.5, \Rz:=2), v200, z200, Tooldata_9;
MoveJ RelTool (starting_position, -156,4, -359.4 \Rx:=4.2, \Ry:=-21.9, \Rz:=1), v200, z200, Tooldata_9;
MoveJ RelTool (starting_position, -151,4, -352.2 \Rx:=4.1, \Ry:=-21.6, \Rz:=1), v200, z200, Tooldata_9;
MoveJ RelTool (starting_position, -146,4, -345.1 \Rx:=4.1, \Ry:=-21, \Rz:=1), v200, z200, Tooldata_9;
MoveJ RelTool (starting_position, -140,4, -338.3 \Rx:=4.1, \Ry:=-20.4, \Rz:=1), v200, z200, Tooldata_9;
MoveJ RelTool (starting_position, -134,4, -331.9 \Rx:=4.1, \Ry:=-19.8, \Rz:=1), v200, z200, Tooldata_9;
MoveJ RelTool (starting_position, -127,4, -326.2 \Rx:=4.1, \Ry:=-19.5, \Rz:=1), v200, z200, Tooldata_9;
MoveJ RelTool (starting_position, -120,4, -321.2 \Rx:=4, \Ry:=-18.9, \Rz:=1), v200, z200, Tooldata_9;
MoveJ RelTool (starting_position, -113,4, -317 \Rx:=4, \Ry:=-18.3, \Rz:=1), v200, z200, Tooldata_9;
MoveJ RelTool (starting_position, -105,4, -313.6 \Rx:=4, \Ry:=-17.4, \Rz:=1), v200, z200, Tooldata_9;
MoveJ RelTool (starting_position, -97,4, -311.1 \Rx:=4, \Ry:=-16.5, \Rz:=1), v200, z200, Tooldata_9;
MoveJ RelTool (starting_position, -89,4, -309.4 \Rx:=4, \Ry:=-15.9, \Rz:=1), v200, z200, Tooldata_9;
MoveJ RelTool (starting_position, -81,4, -308.1 \Rx:=3.9, \Ry:=-15.3, \Rz:=1), v200, z200, Tooldata_9;
MoveJ RelTool (starting_position, -73,4, -307.4 \Rx:=3.9, \Ry:=-14.4, \Rz:=1), v200, z200, Tooldata_9;
MoveJ RelTool (starting_position, -65,4, -307.1 \Rx:=3.9, \Ry:=-13.8, \Rz:=1), v200, z200, Tooldata_9;
MoveJ RelTool (starting_position, -57,0, -307.1 \Rx:=3.9, \Ry:=-12.9, \Rz:=0), v200, z200, Tooldata_9;
MoveJ RelTool (starting_position, -50,0, -307.2 \Rx:=3.9, \Ry:=-12.3, \Rz:=0), v200, z200, Tooldata_9;
MoveJ RelTool (starting_position, -43,0, -307.4 \Rx:=3.8, \Ry:=-11.4, \Rz:=0), v200, z200, Tooldata_9;
MoveJ RelTool (starting_position, -36,0, -307.5 \Rx:=3.8, \Ry:=-10.8, \Rz:=0), v200, z200, Tooldata_9;
MoveJ RelTool (starting_position, -29,0, -307.7 \Rx:=3.8, \Ry:=-10.5, \Rz:=0), v200, z200, Tooldata_9;
MoveJ RelTool (starting_position, -23,0, -307.9 \Rx:=3.8, \Ry:=-9.9, \Rz:=0), v200, z200, Tooldata_9;
MoveJ RelTool (starting_position, -18,0, -308 \Rx:=3.8, \Ry:=-9.6, \Rz:=0), v200, z200, Tooldata_9;
MoveJ RelTool (starting_position, -12,-0, -308.1 \Rx:=3.8, \Ry:=-9, \Rz:=-0), v200, z200, Tooldata_9;
MoveJ RelTool (starting_position, -8,-0, -308.5 \Rx:=3.8, \Ry:=-8.4, \Rz:=-0), v200, z200, Tooldata_9;
MoveJ RelTool (starting_position, -4,-0, -309 \Rx:=3.8, \Ry:=-8.1, \Rz:=-0), v200, z200, Tooldata_9;
MoveJ RelTool (starting_position, 0,-0, -309.7 \Rx:=3.8, \Ry:=-7.8, \Rz:=-0), v200, z200, Tooldata_9;
MoveJ RelTool (starting_position, 3,-0, -310.6 \Rx:=3.8, \Ry:=-7.5, \Rz:=-0), v200, z200, Tooldata_9;
MoveJ RelTool (starting_position, 6,-0, -311.8 \Rx:=3.8, \Ry:=-7.5, \Rz:=-0), v200, z200, Tooldata_9;
MoveJ RelTool (starting_position, 8,-4, -313.1 \Rx:=3.8, \Ry:=-7.2, \Rz:=-1), v200, z200, Tooldata_9;
MoveJ RelTool (starting_position, 9,-4, -314.4 \Rx:=3.8, \Ry:=-7.2, \Rz:=-1), v200, z200, Tooldata_9;
MoveJ RelTool (starting_position, 10,-4, -315.5 \Rx:=3.8, \Ry:=-6.9, \Rz:=-1), v200, z200, Tooldata_9;
MoveJ RelTool (starting_position, 11,-4, -316.5 \Rx:=3.8, \Ry:=-6.9, \Rz:=-1), v200, z200, Tooldata_9;
MoveJ RelTool (starting_position, 11,-4, -317.1 \Rx:=3.8, \Ry:=-6.9, \Rz:=-1), v200, z200, Tooldata_9;
MoveJ RelTool (starting_position, 11,-4, -317.3 \Rx:=3.8, \Ry:=-6.9, \Rz:=-1), v200, z200, Tooldata_9;
MoveJ RelTool (starting_position, 11,-4, -317.1 \Rx:=3.8, \Ry:=-7.2, \Rz:=-1), v200, z200, Tooldata_9;
MoveJ RelTool (starting_position, 10,-4, -316.5 \Rx:=3.9, \Ry:=-7.2, \Rz:=-1), v200, z200, Tooldata_9;
MoveJ RelTool (starting_position, 9,-4, -315.5 \Rx:=3.9, \Ry:=-7.2, \Rz:=-1), v200, z200, Tooldata_9;
MoveJ RelTool (starting_position, 8,-4, -314 \Rx:=3.9, \Ry:=-7.5, \Rz:=-1), v200, z200, Tooldata_9;
MoveJ RelTool (starting_position, 6,-4, -312.2 \Rx:=4, \Ry:=-7.5, \Rz:=-1), v200, z200, Tooldata_9;
MoveJ RelTool (starting_position, 5,-4, -310 \Rx:=4, \Ry:=-7.8, \Rz:=-1), v200, z200, Tooldata_9;
MoveJ RelTool (starting_position, 3,-4, -307.5 \Rx:=4, \Ry:=-7.8, \Rz:=-1), v200, z200, Tooldata_9;
MoveJ RelTool (starting_position, 1,-4, -304.6 \Rx:=4.1, \Ry:=-8.1, \Rz:=-1), v200, z200, Tooldata_9;
MoveJ RelTool (starting_position, -1,-8, -301.5 \Rx:=4.1, \Ry:=-8.1, \Rz:=-2), v200, z200, Tooldata_9;
MoveJ RelTool (starting_position, -3,-8, -298.2 \Rx:=4.2, \Ry:=-8.4, \Rz:=-2), v200, z200, Tooldata_9;
MoveJ RelTool (starting_position, -5,-8, -295 \Rx:=4.2, \Ry:=-8.7, \Rz:=-2), v200, z200, Tooldata_9;
MoveJ RelTool (starting_position, -8,-8, -291.9 \Rx:=4.2, \Ry:=-9, \Rz:=-2), v200, z200, Tooldata_9;
MoveJ RelTool (starting_position, -10,-8, -289.1 \Rx:=4.3, \Ry:=-9, \Rz:=-2), v200, z200, Tooldata_9;
MoveJ RelTool (starting_position, -13,-8, -286.6 \Rx:=4.3, \Ry:=-9.3, \Rz:=-2), v200, z200, Tooldata_9;
MoveJ RelTool (starting_position, -15,-8, -284.6 \Rx:=4.3, \Ry:=-9.3, \Rz:=-2), v200, z200, Tooldata_9;
MoveJ RelTool (starting_position, -18,-8, -282.9 \Rx:=4.4, \Ry:=-9.6, \Rz:=-2), v200, z200, Tooldata_9;
MoveJ RelTool (starting_position, -21,-8, -281.6 \Rx:=4.4, \Ry:=-9.9, \Rz:=-2), v200, z200, Tooldata_9;
MoveJ RelTool (starting_position, -23,-8, -280.5 \Rx:=4.5, \Ry:=-10.2, \Rz:=-2), v200, z200, Tooldata_9;
MoveJ RelTool (starting_position, -26,-8, -279.6 \Rx:=4.5, \Ry:=-10.5, \Rz:=-2), v200, z200, Tooldata_9;
MoveJ RelTool (starting_position, -29,-8, -278.7 \Rx:=4.6, \Ry:=-10.8, \Rz:=-2), v200, z200, Tooldata_9;
MoveJ RelTool (starting_position, -32,-8, -277.8 \Rx:=4.7, \Ry:=-11.1, \Rz:=-2), v200, z200, Tooldata_9;
MoveJ RelTool (starting_position, -35,-12, -276.8 \Rx:=4.7, \Ry:=-11.1, \Rz:=-3), v200, z200, Tooldata_9;
MoveJ RelTool (starting_position, -38,-12, -275.6 \Rx:=4.8, \Ry:=-11.4, \Rz:=-3), v200, z200, Tooldata_9;
MoveJ RelTool (starting_position, -41,-12, -274.2 \Rx:=4.9, \Ry:=-11.7, \Rz:=-3), v200, z200, Tooldata_9;
MoveJ RelTool (starting_position, -44,-12, -272.6 \Rx:=4.9, \Ry:=-12, \Rz:=-3), v200, z200, Tooldata_9;
MoveJ RelTool (starting_position, -47,-12, -271 \Rx:=5, \Ry:=-12.3, \Rz:=-3), v200, z200, Tooldata_9;
MoveJ RelTool (starting_position, -50,-12, -269.3 \Rx:=5.1, \Ry:=-12.6, \Rz:=-3), v200, z200, Tooldata_9;
MoveJ RelTool (starting_position, -53,-12, -267.7 \Rx:=5.1, \Ry:=-12.6, \Rz:=-3), v200, z200, Tooldata_9;
MoveJ RelTool (starting_position, -57,-12, -266.2 \Rx:=5.2, \Ry:=-13.2, \Rz:=-3), v200, z200, Tooldata_9;
MoveJ RelTool (starting_position, -60,-12, -264.9 \Rx:=5.3, \Ry:=-13.2, \Rz:=-3), v200, z200, Tooldata_9;
MoveJ RelTool (starting_position, -64,-12, -263.6 \Rx:=5.3, \Ry:=-13.5, \Rz:=-3), v200, z200, Tooldata_9;
MoveJ RelTool (starting_position, -67,-12, -262.3 \Rx:=5.4, \Ry:=-13.8, \Rz:=-3), v200, z200, Tooldata_9;
MoveJ RelTool (starting_position, -71,-12, -261 \Rx:=5.5, \Ry:=-14.4, \Rz:=-3), v200, z200, Tooldata_9;
MoveJ RelTool (starting_position, -75,-12, -259.6 \Rx:=5.6, \Ry:=-14.7, \Rz:=-3), v200, z200, Tooldata_9;
MoveJ RelTool (starting_position, -79,-12, -258.1 \Rx:=5.6, \Ry:=-15, \Rz:=-3), v200, z200, Tooldata_9;
MoveJ RelTool (starting_position, -84,-16, -256.5 \Rx:=5.7, \Ry:=-15.3, \Rz:=-4), v200, z200, Tooldata_9;
MoveJ RelTool (starting_position, -88,-16, -254.7 \Rx:=5.8, \Ry:=-15.6, \Rz:=-4), v200, z200, Tooldata_9;
MoveJ RelTool (starting_position, -92,-16, -252.7 \Rx:=5.9, \Ry:=-16.2, \Rz:=-4), v200, z200, Tooldata_9;
MoveJ RelTool (starting_position, -97,-16, -250.5 \Rx:=6, \Ry:=-16.8, \Rz:=-4), v200, z200, Tooldata_9;
MoveJ RelTool (starting_position, -101,-16, -248.2 \Rx:=6.1, \Ry:=-17.1, \Rz:=-4), v200, z200, Tooldata_9;
MoveJ RelTool (starting_position, -106,-16, -245.6 \Rx:=6.1, \Ry:=-17.4, \Rz:=-4), v200, z200, Tooldata_9;
MoveJ RelTool (starting_position, -110,-16, -243 \Rx:=6.2, \Ry:=-17.7, \Rz:=-4), v200, z200, Tooldata_9;
MoveJ RelTool (starting_position, -115,-16, -240.2 \Rx:=6.3, \Ry:=-18, \Rz:=-4), v200, z200, Tooldata_9;
MoveJ RelTool (starting_position, -119,-16, -237.4 \Rx:=6.4, \Ry:=-18.6, \Rz:=-4), v200, z200, Tooldata_9;
MoveJ RelTool (starting_position, -124,-16, -234.6 \Rx:=6.5, \Ry:=-18.9, \Rz:=-4), v200, z200, Tooldata_9;
MoveJ RelTool (starting_position, -128,-16, -231.8 \Rx:=6.6, \Ry:=-19.2, \Rz:=-4), v200, z200, Tooldata_9;
MoveJ RelTool (starting_position, -132,-16, -229 \Rx:=6.7, \Ry:=-19.8, \Rz:=-4), v200, z200, Tooldata_9;
MoveJ RelTool (starting_position, -137,-16, -226 \Rx:=6.8, \Ry:=-20.1, \Rz:=-4), v200, z200, Tooldata_9;
MoveJ RelTool (starting_position, -141,-16, -223 \Rx:=6.9, \Ry:=-20.4, \Rz:=-4), v200, z200, Tooldata_9;
MoveJ RelTool (starting_position, -145,-20, -219.8 \Rx:=7, \Ry:=-20.7, \Rz:=-5), v200, z200, Tooldata_9;
MoveJ RelTool (starting_position, -149,-20, -216.4 \Rx:=7.1, \Ry:=-21.3, \Rz:=-5), v200, z200, Tooldata_9;
MoveJ RelTool (starting_position, -153,-20, -213 \Rx:=7.1, \Ry:=-21.6, \Rz:=-5), v200, z200, Tooldata_9;
MoveJ RelTool (starting_position, -157,-20, -209.3 \Rx:=7.2, \Ry:=-21.6, \Rz:=-5), v200, z200, Tooldata_9;
MoveJ RelTool (starting_position, -160,-20, -205.5 \Rx:=7.3, \Ry:=-22.2, \Rz:=-5), v200, z200, Tooldata_9;
MoveJ RelTool (starting_position, -164,-20, -201.6 \Rx:=7.4, \Ry:=-22.5, \Rz:=-5), v200, z200, Tooldata_9;
MoveJ RelTool (starting_position, -167,-20, -197.6 \Rx:=7.5, \Ry:=-22.8, \Rz:=-5), v200, z200, Tooldata_9;
MoveJ RelTool (starting_position, -170,-20, -193.5 \Rx:=7.6, \Ry:=-23.1, \Rz:=-5), v200, z200, Tooldata_9;
MoveJ RelTool (starting_position, -173,-20, -189.4 \Rx:=7.7, \Ry:=-23.4, \Rz:=-5), v200, z200, Tooldata_9;
MoveJ RelTool (starting_position, -175,-20, -185.2 \Rx:=7.8, \Ry:=-23.4, \Rz:=-5), v200, z200, Tooldata_9;
MoveJ RelTool (starting_position, -178,-20, -181 \Rx:=7.9, \Ry:=-23.7, \Rz:=-5), v200, z200, Tooldata_9;
MoveJ RelTool (starting_position, -180,-20, -176.9 \Rx:=8, \Ry:=-24, \Rz:=-5), v200, z200, Tooldata_9;
MoveJ RelTool (starting_position, -182,-20, -172.8 \Rx:=8.1, \Ry:=-24, \Rz:=-5), v200, z200, Tooldata_9;
MoveJ RelTool (starting_position, -183,-20, -168.7 \Rx:=8.1, \Ry:=-24.3, \Rz:=-5), v200, z200, Tooldata_9;
MoveJ RelTool (starting_position, -185,-24, -164.5 \Rx:=8.2, \Ry:=-24.3, \Rz:=-6), v200, z200, Tooldata_9;
MoveJ RelTool (starting_position, -186,-24, -160.4 \Rx:=8.3, \Ry:=-24.3, \Rz:=-6), v200, z200, Tooldata_9;
MoveJ RelTool (starting_position, -187,-24, -156.2 \Rx:=8.4, \Ry:=-24.6, \Rz:=-6), v200, z200, Tooldata_9;
MoveJ RelTool (starting_position, -188,-24, -152.1 \Rx:=8.5, \Ry:=-24.6, \Rz:=-6), v200, z200, Tooldata_9;
MoveJ RelTool (starting_position, -188,-24, -148 \Rx:=8.5, \Ry:=-24.6, \Rz:=-6), v200, z200, Tooldata_9;
MoveJ RelTool (starting_position, -188,-24, -143.9 \Rx:=8.6, \Ry:=-24.6, \Rz:=-6), v200, z200, Tooldata_9;
MoveJ RelTool (starting_position, -188,-24, -139.7 \Rx:=8.7, \Ry:=-24.6, \Rz:=-6), v200, z200, Tooldata_9;
MoveJ RelTool (starting_position, -188,-24, -135.6 \Rx:=8.8, \Ry:=-24.6, \Rz:=-6), v200, z200, Tooldata_9;
MoveJ RelTool (starting_position, -188,-24, -131.5 \Rx:=8.9, \Ry:=-24.6, \Rz:=-6), v200, z200, Tooldata_9;
MoveJ RelTool (starting_position, -187,-24, -127.4 \Rx:=9, \Ry:=-24.6, \Rz:=-6), v200, z200, Tooldata_9;
MoveJ RelTool (starting_position, -186,-24, -123.3 \Rx:=9, \Ry:=-24.3, \Rz:=-6), v200, z200, Tooldata_9;
MoveJ RelTool (starting_position, -185,-24, -119.1 \Rx:=9.1, \Ry:=-24.3, \Rz:=-6), v200, z200, Tooldata_9;
MoveJ RelTool (starting_position, -184,-24, -114.9 \Rx:=9.2, \Ry:=-24.3, \Rz:=-6), v200, z200, Tooldata_9;
MoveJ RelTool (starting_position, -183,-24, -110.7 \Rx:=9.2, \Ry:=-24, \Rz:=-6), v200, z200, Tooldata_9;
MoveJ RelTool (starting_position, -181,-28, -106.6 \Rx:=9.3, \Ry:=-24, \Rz:=-7), v200, z200, Tooldata_9;
MoveJ RelTool (starting_position, -180,-28, -102.6 \Rx:=9.4, \Ry:=-23.7, \Rz:=-7), v200, z200, Tooldata_9;
MoveJ RelTool (starting_position, -178,-28, -98.6 \Rx:=9.4, \Ry:=-23.7, \Rz:=-7), v200, z200, Tooldata_9;
MoveJ RelTool (starting_position, -176,-28, -94.9 \Rx:=9.5, \Ry:=-23.4, \Rz:=-7), v200, z200, Tooldata_9;
MoveJ RelTool (starting_position, -175,-28, -91.2 \Rx:=9.6, \Ry:=-23.4, \Rz:=-7), v200, z200, Tooldata_9;
MoveJ RelTool (starting_position, -173,-28, -87.7 \Rx:=9.6, \Ry:=-23.1, \Rz:=-7), v200, z200, Tooldata_9;
MoveJ RelTool (starting_position, -171,-28, -84.4 \Rx:=9.7, \Ry:=-23.1, \Rz:=-7), v200, z200, Tooldata_9;
MoveJ RelTool (starting_position, -169,-28, -81.1 \Rx:=9.7, \Ry:=-22.8, \Rz:=-7), v200, z200, Tooldata_9;
MoveJ RelTool (starting_position, -167,-28, -78 \Rx:=9.8, \Ry:=-22.5, \Rz:=-7), v200, z200, Tooldata_9;
MoveJ RelTool (starting_position, -165,-28, -75.1 \Rx:=9.8, \Ry:=-22.5, \Rz:=-7), v200, z200, Tooldata_9;
MoveJ RelTool (starting_position, -163,-28, -72.3 \Rx:=9.9, \Ry:=-22.2, \Rz:=-7), v200, z200, Tooldata_9;
MoveJ RelTool (starting_position, -161,-28, -69.6 \Rx:=9.9, \Ry:=-22.2, \Rz:=-7), v200, z200, Tooldata_9;
MoveJ RelTool (starting_position, -160,-28, -67.2 \Rx:=9.9, \Ry:=-22.2, \Rz:=-7), v200, z200, Tooldata_9;
MoveJ RelTool (starting_position, -158,-28, -64.9 \Rx:=10, \Ry:=-21.9, \Rz:=-7), v200, z200, Tooldata_9;
MoveJ RelTool (starting_position, -156,-28, -62.5 \Rx:=10, \Ry:=-21.6, \Rz:=-7), v200, z200, Tooldata_9;
MoveJ RelTool (starting_position, -153,-28, -60.1 \Rx:=10.1, \Ry:=-21.3, \Rz:=-7), v200, z200, Tooldata_9;
MoveJ RelTool (starting_position, -151,-32, -57.5 \Rx:=10.1, \Ry:=-21.3, \Rz:=-8), v200, z200, Tooldata_9;
MoveJ RelTool (starting_position, -149,-32, -54.8 \Rx:=10.2, \Ry:=-21.3, \Rz:=-8), v200, z200, Tooldata_9;
MoveJ RelTool (starting_position, -147,-32, -51.8 \Rx:=10.2, \Ry:=-21, \Rz:=-8), v200, z200, Tooldata_9;
MoveJ RelTool (starting_position, -145,-32, -48.6 \Rx:=10.3, \Ry:=-20.7, \Rz:=-8), v200, z200, Tooldata_9;
MoveJ RelTool (starting_position, -143,-32, -45.2 \Rx:=10.3, \Ry:=-20.4, \Rz:=-8), v200, z200, Tooldata_9;
MoveJ RelTool (starting_position, -141,-32, -41.6 \Rx:=10.3, \Ry:=-20.4, \Rz:=-8), v200, z200, Tooldata_9;
MoveJ RelTool (starting_position, -139,-32, -37.9 \Rx:=10.4, \Ry:=-20.1, \Rz:=-8), v200, z200, Tooldata_9;
MoveJ RelTool (starting_position, -137,-32, -34.2 \Rx:=10.4, \Ry:=-20.1, \Rz:=-8), v200, z200, Tooldata_9;
MoveJ RelTool (starting_position, -134,-32, -30.5 \Rx:=10.4, \Ry:=-19.8, \Rz:=-8), v200, z200, Tooldata_9;
MoveJ RelTool (starting_position, -132,-32, -26.7 \Rx:=10.4, \Ry:=-19.8, \Rz:=-8), v200, z200, Tooldata_9;
MoveJ RelTool (starting_position, -130,-32, -23 \Rx:=10.4, \Ry:=-19.5, \Rz:=-8), v200, z200, Tooldata_9;
MoveJ RelTool (starting_position, -127,-32, -19.3 \Rx:=10.4, \Ry:=-19.2, \Rz:=-8), v200, z200, Tooldata_9;
MoveJ RelTool (starting_position, -125,-32, -15.7 \Rx:=10.4, \Ry:=-18.9, \Rz:=-8), v200, z200, Tooldata_9;
MoveJ RelTool (starting_position, -122,-32, -12.2 \Rx:=10.4, \Ry:=-18.9, \Rz:=-8), v200, z200, Tooldata_9;
MoveJ RelTool (starting_position, -120,-32, -8.8 \Rx:=10.4, \Ry:=-18.6, \Rz:=-8), v200, z200, Tooldata_9;
MoveJ RelTool (starting_position, -117,-36, -5.5 \Rx:=10.4, \Ry:=-18.3, \Rz:=-9), v200, z200, Tooldata_9;
MoveJ RelTool (starting_position, -115,-36, -2.4 \Rx:=10.4, \Ry:=-18, \Rz:=-9), v200, z200, Tooldata_9;
MoveJ RelTool (starting_position, -112,-36, 0.6 \Rx:=10.4, \Ry:=-18, \Rz:=-9), v200, z200, Tooldata_9;
MoveJ RelTool (starting_position, -110,-36, 3.4 \Rx:=10.4, \Ry:=-17.7, \Rz:=-9), v200, z200, Tooldata_9;
MoveJ RelTool (starting_position, -107,-36, 6.1 \Rx:=10.4, \Ry:=-17.4, \Rz:=-9), v200, z200, Tooldata_9;
MoveJ RelTool (starting_position, -104,-36, 8.6 \Rx:=10.4, \Ry:=-17.4, \Rz:=-9), v200, z200, Tooldata_9;
MoveJ RelTool (starting_position, -101,-36, 10.9 \Rx:=10.4, \Ry:=-17.1, \Rz:=-9), v200, z200, Tooldata_9;
MoveJ RelTool (starting_position, -98,-36, 13.1 \Rx:=10.4, \Ry:=-16.8, \Rz:=-9), v200, z200, Tooldata_9;
MoveJ RelTool (starting_position, -95,-36, 15.3 \Rx:=10.4, \Ry:=-16.5, \Rz:=-9), v200, z200, Tooldata_9;
MoveJ RelTool (starting_position, -92,-36, 17.4 \Rx:=10.4, \Ry:=-16.2, \Rz:=-9), v200, z200, Tooldata_9;
MoveJ RelTool (starting_position, -89,-36, 19.6 \Rx:=10.4, \Ry:=-15.9, \Rz:=-9), v200, z200, Tooldata_9;
MoveJ RelTool (starting_position, -86,-36, 21.9 \Rx:=10.4, \Ry:=-15.6, \Rz:=-9), v200, z200, Tooldata_9;
MoveJ RelTool (starting_position, -82,-36, 24.3 \Rx:=10.4, \Ry:=-15.3, \Rz:=-9), v200, z200, Tooldata_9;
MoveJ RelTool (starting_position, -79,-36, 26.8 \Rx:=10.3, \Ry:=-15, \Rz:=-9), v200, z200, Tooldata_9;
MoveJ RelTool (starting_position, -75,-36, 29.2 \Rx:=10.3, \Ry:=-14.7, \Rz:=-9), v200, z200, Tooldata_9;
MoveJ RelTool (starting_position, -72,-36, 31.5 \Rx:=10.3, \Ry:=-14.4, \Rz:=-9), v200, z200, Tooldata_9;
MoveJ RelTool (starting_position, -69,-36, 33.8 \Rx:=10.3, \Ry:=-14.1, \Rz:=-9), v200, z200, Tooldata_9;
MoveJ RelTool (starting_position, -65,-40, 36.1 \Rx:=10.3, \Ry:=-13.8, \Rz:=-10), v200, z200, Tooldata_9;
MoveJ RelTool (starting_position, -62,-40, 38.3 \Rx:=10.3, \Ry:=-13.5, \Rz:=-10), v200, z200, Tooldata_9;
MoveJ RelTool (starting_position, -58,-40, 40.3 \Rx:=10.3, \Ry:=-13.2, \Rz:=-10), v200, z200, Tooldata_9;
MoveJ RelTool (starting_position, -55,-40, 42.3 \Rx:=10.2, \Ry:=-12.9, \Rz:=-10), v200, z200, Tooldata_9;
MoveJ RelTool (starting_position, -52,-40, 44.1 \Rx:=10.2, \Ry:=-12.6, \Rz:=-10), v200, z200, Tooldata_9;
MoveJ RelTool (starting_position, -49,-40, 45.9 \Rx:=10.2, \Ry:=-12.3, \Rz:=-10), v200, z200, Tooldata_9;
MoveJ RelTool (starting_position, -46,-40, 47.7 \Rx:=10.2, \Ry:=-12, \Rz:=-10), v200, z200, Tooldata_9;
MoveJ RelTool (starting_position, -43,-40, 49.5 \Rx:=10.2, \Ry:=-12, \Rz:=-10), v200, z200, Tooldata_9;
MoveJ RelTool (starting_position, -39,-40, 51.3 \Rx:=10.2, \Ry:=-11.7, \Rz:=-10), v200, z200, Tooldata_9;
MoveJ RelTool (starting_position, -36,-40, 53.1 \Rx:=10.2, \Ry:=-11.4, \Rz:=-10), v200, z200, Tooldata_9;
MoveJ RelTool (starting_position, -33,-40, 55 \Rx:=10.2, \Ry:=-11.1, \Rz:=-10), v200, z200, Tooldata_9;
MoveJ RelTool (starting_position, -30,-40, 56.9 \Rx:=10.2, \Ry:=-10.8, \Rz:=-10), v200, z200, Tooldata_9;
MoveJ RelTool (starting_position, -27,-40, 58.9 \Rx:=10.2, \Ry:=-10.5, \Rz:=-10), v200, z200, Tooldata_9;
MoveJ RelTool (starting_position, -23,-40, 61 \Rx:=10.2, \Ry:=-10.2, \Rz:=-10), v200, z200, Tooldata_9;
MoveJ RelTool (starting_position, -20,-40, 62.9 \Rx:=10.2, \Ry:=-9.9, \Rz:=-10), v200, z200, Tooldata_9;
MoveJ RelTool (starting_position, -16,-40, 64.8 \Rx:=10.2, \Ry:=-9.6, \Rz:=-10), v200, z200, Tooldata_9;
MoveJ RelTool (starting_position, -13,-40, 66.6 \Rx:=10.2, \Ry:=-9.3, \Rz:=-10), v200, z200, Tooldata_9;
MoveJ RelTool (starting_position, -10,-40, 68.3 \Rx:=10.2, \Ry:=-9, \Rz:=-10), v200, z200, Tooldata_9;
MoveJ RelTool (starting_position, -6,-44, 69.7 \Rx:=10.3, \Ry:=-8.7, \Rz:=-11), v200, z200, Tooldata_9;
MoveJ RelTool (starting_position, -3,-44, 71 \Rx:=10.3, \Ry:=-8.4, \Rz:=-11), v200, z200, Tooldata_9;
MoveJ RelTool (starting_position, 0,-44, 72.2 \Rx:=10.3, \Ry:=-8.1, \Rz:=-11), v200, z200, Tooldata_9;
MoveJ RelTool (starting_position, 3,-44, 73.4 \Rx:=10.3, \Ry:=-7.8, \Rz:=-11), v200, z200, Tooldata_9;
MoveJ RelTool (starting_position, 5,-44, 74.6 \Rx:=10.3, \Ry:=-7.5, \Rz:=-11), v200, z200, Tooldata_9;
MoveJ RelTool (starting_position, 8,-44, 76 \Rx:=10.4, \Ry:=-7.5, \Rz:=-11), v200, z200, Tooldata_9;
MoveJ RelTool (starting_position, 11,-44, 77.4 \Rx:=10.4, \Ry:=-7.2, \Rz:=-11), v200, z200, Tooldata_9;
MoveJ RelTool (starting_position, 13,-44, 78.7 \Rx:=10.4, \Ry:=-6.9, \Rz:=-11), v200, z200, Tooldata_9;
MoveJ RelTool (starting_position, 15,-44, 80.1 \Rx:=10.4, \Ry:=-6.9, \Rz:=-11), v200, z200, Tooldata_9;
MoveJ RelTool (starting_position, 17,-44, 81.1 \Rx:=10.5, \Ry:=-6.6, \Rz:=-11), v200, z200, Tooldata_9;
MoveJ RelTool (starting_position, 19,-44, 81.9 \Rx:=10.5, \Ry:=-6.6, \Rz:=-11), v200, z200, Tooldata_9;
MoveJ RelTool (starting_position, 21,-44, 82.1 \Rx:=10.6, \Ry:=-6.3, \Rz:=-11), v200, z200, Tooldata_9;
MoveJ RelTool (starting_position, 23,-44, 81.9 \Rx:=10.6, \Ry:=-6, \Rz:=-11), v200, z200, Tooldata_9;
MoveJ RelTool (starting_position, 25,-44, 81 \Rx:=10.7, \Ry:=-6, \Rz:=-11), v200, z200, Tooldata_9;
MoveJ RelTool (starting_position, 26,-44, 79.8 \Rx:=10.7, \Ry:=-5.7, \Rz:=-11), v200, z200, Tooldata_9;
MoveJ RelTool (starting_position, 28,-44, 78.2 \Rx:=10.8, \Ry:=-5.7, \Rz:=-11), v200, z200, Tooldata_9;
MoveJ RelTool (starting_position, 29,-44, 76.6 \Rx:=10.8, \Ry:=-5.7, \Rz:=-11), v200, z200, Tooldata_9;
MoveJ RelTool (starting_position, 31,-44, 75.1 \Rx:=10.9, \Ry:=-5.4, \Rz:=-11), v200, z200, Tooldata_9;
MoveJ RelTool (starting_position, 32,-44, 73.8 \Rx:=11, \Ry:=-5.4, \Rz:=-11), v200, z200, Tooldata_9;
MoveJ RelTool (starting_position, 33,-44, 73 \Rx:=11, \Ry:=-5.4, \Rz:=-11), v200, z200, Tooldata_9;
MoveJ RelTool (starting_position, 34,-48, 72.8 \Rx:=11.1, \Ry:=-5.1, \Rz:=-12), v200, z200, Tooldata_9;
MoveJ RelTool (starting_position, 36,-48, 73.3 \Rx:=11.2, \Ry:=-5.1, \Rz:=-12), v200, z200, Tooldata_9;
MoveJ RelTool (starting_position, 37,-48, 74.5 \Rx:=11.3, \Ry:=-5.1, \Rz:=-12), v200, z200, Tooldata_9;
MoveJ RelTool (starting_position, 38,-48, 76.3 \Rx:=11.3, \Ry:=-5.1, \Rz:=-12), v200, z200, Tooldata_9;
MoveJ RelTool (starting_position, 40,-48, 78.7 \Rx:=11.4, \Ry:=-4.8, \Rz:=-12), v200, z200, Tooldata_9;
MoveJ RelTool (starting_position, 41,-48, 81.4 \Rx:=11.5, \Ry:=-4.5, \Rz:=-12), v200, z200, Tooldata_9;
MoveJ RelTool (starting_position, 43,-48, 84.5 \Rx:=11.6, \Ry:=-4.5, \Rz:=-12), v200, z200, Tooldata_9;
MoveJ RelTool (starting_position, 44,-48, 87.6 \Rx:=11.6, \Ry:=-4.5, \Rz:=-12), v200, z200, Tooldata_9;
MoveJ RelTool (starting_position, 46,-48, 90.7 \Rx:=11.7, \Ry:=-4.2, \Rz:=-12), v200, z200, Tooldata_9;
MoveJ RelTool (starting_position, 48,-48, 93.7 \Rx:=11.8, \Ry:=-4.2, \Rz:=-12), v200, z200, Tooldata_9;
MoveJ RelTool (starting_position, 50,-48, 96.3 \Rx:=11.9, \Ry:=-3.9, \Rz:=-12), v200, z200, Tooldata_9;
MoveJ RelTool (starting_position, 53,-48, 98.5 \Rx:=12, \Ry:=-3.9, \Rz:=-12), v200, z200, Tooldata_9;
MoveJ RelTool (starting_position, 55,-48, 100.2 \Rx:=12.1, \Ry:=-3.6, \Rz:=-12), v200, z200, Tooldata_9;
MoveJ RelTool (starting_position, 58,-48, 101.4 \Rx:=12.1, \Ry:=-3.3, \Rz:=-12), v200, z200, Tooldata_9;
MoveJ RelTool (starting_position, 61,-48, 102 \Rx:=12.2, \Ry:=-3, \Rz:=-12), v200, z200, Tooldata_9;
MoveJ RelTool (starting_position, 64,-48, 102.1 \Rx:=12.3, \Ry:=-3, \Rz:=-12), v200, z200, Tooldata_9;
MoveJ RelTool (starting_position, 68,-48, 101.7 \Rx:=12.4, \Ry:=-2.4, \Rz:=-12), v200, z200, Tooldata_9;
MoveJ RelTool (starting_position, 72,-48, 100.9 \Rx:=12.5, \Ry:=-2.1, \Rz:=-12), v200, z200, Tooldata_9;
MoveJ RelTool (starting_position, 76,-48, 99.8 \Rx:=12.6, \Ry:=-1.8, \Rz:=-12), v200, z200, Tooldata_9;
MoveJ RelTool (starting_position, 80,-48, 98.7 \Rx:=12.7, \Ry:=-1.2, \Rz:=-12), v200, z200, Tooldata_9;
MoveJ RelTool (starting_position, 84,-48, 97.6 \Rx:=12.8, \Ry:=-0.9, \Rz:=-12), v200, z200, Tooldata_9;
MoveJ RelTool (starting_position, 88,-48, 96.6 \Rx:=12.9, \Ry:=-0.6, \Rz:=-12), v200, z200, Tooldata_9;
MoveJ RelTool (starting_position, 93,-52, 95.9 \Rx:=13, \Ry:=-0, \Rz:=-13), v200, z200, Tooldata_9;
MoveJ RelTool (starting_position, 97,-52, 95.6 \Rx:=13.1, \Ry:=0.3, \Rz:=-13), v200, z200, Tooldata_9;
MoveJ RelTool (starting_position, 101,-52, 95.5 \Rx:=13.2, \Ry:=0.6, \Rz:=-13), v200, z200, Tooldata_9;
MoveJ RelTool (starting_position, 105,-52, 95.8 \Rx:=13.3, \Ry:=0.9, \Rz:=-13), v200, z200, Tooldata_9;
MoveJ RelTool (starting_position, 110,-52, 96.2 \Rx:=13.3, \Ry:=1.2, \Rz:=-13), v200, z200, Tooldata_9;
MoveJ RelTool (starting_position, 114,-52, 96.8 \Rx:=13.4, \Ry:=1.5, \Rz:=-13), v200, z200, Tooldata_9;
MoveJ RelTool (starting_position, 118,-52, 97.4 \Rx:=13.5, \Ry:=2.1, \Rz:=-13), v200, z200, Tooldata_9;
MoveJ RelTool (starting_position, 123,-52, 98 \Rx:=13.6, \Ry:=2.4, \Rz:=-13), v200, z200, Tooldata_9;
MoveJ RelTool (starting_position, 128,-52, 98.4 \Rx:=13.7, \Ry:=2.7, \Rz:=-13), v200, z200, Tooldata_9;
MoveJ RelTool (starting_position, 132,-52, 98.7 \Rx:=13.8, \Ry:=3.3, \Rz:=-13), v200, z200, Tooldata_9;
MoveJ RelTool (starting_position, 137,-52, 98.9 \Rx:=13.8, \Ry:=3.6, \Rz:=-13), v200, z200, Tooldata_9;
MoveJ RelTool (starting_position, 142,-52, 99.3 \Rx:=13.9, \Ry:=3.9, \Rz:=-13), v200, z200, Tooldata_9;
MoveJ RelTool (starting_position, 147,-52, 99.8 \Rx:=13.9, \Ry:=4.5, \Rz:=-13), v200, z200, Tooldata_9;
MoveJ RelTool (starting_position, 153,-52, 100.5 \Rx:=14, \Ry:=5.1, \Rz:=-13), v200, z200, Tooldata_9;
MoveJ RelTool (starting_position, 158,-52, 101.2 \Rx:=14.1, \Ry:=5.4, \Rz:=-13), v200, z200, Tooldata_9;
MoveJ RelTool (starting_position, 163,-52, 101.9 \Rx:=14.1, \Ry:=6, \Rz:=-13), v200, z200, Tooldata_9;
MoveJ RelTool (starting_position, 169,-52, 102.6 \Rx:=14.2, \Ry:=6.3, \Rz:=-13), v200, z200, Tooldata_9;
MoveJ RelTool (starting_position, 174,-52, 102.9 \Rx:=14.3, \Ry:=6.9, \Rz:=-13), v200, z200, Tooldata_9;
MoveJ RelTool (starting_position, 179,-52, 102.8 \Rx:=14.4, \Ry:=7.5, \Rz:=-13), v200, z200, Tooldata_9;
MoveJ RelTool (starting_position, 184,-52, 102.2 \Rx:=14.4, \Ry:=7.8, \Rz:=-13), v200, z200, Tooldata_9;
MoveJ RelTool (starting_position, 189,-52, 101.3 \Rx:=14.4, \Ry:=8.4, \Rz:=-13), v200, z200, Tooldata_9;
MoveJ RelTool (starting_position, 193,-52, 99.8 \Rx:=14.5, \Ry:=9, \Rz:=-13), v200, z200, Tooldata_9;
MoveJ RelTool (starting_position, 197,-52, 97.9 \Rx:=14.5, \Ry:=9.3, \Rz:=-13), v200, z200, Tooldata_9;
MoveJ RelTool (starting_position, 201,-52, 95.7 \Rx:=14.5, \Ry:=9.6, \Rz:=-13), v200, z200, Tooldata_9;
MoveJ RelTool (starting_position, 204,-52, 93.3 \Rx:=14.6, \Ry:=9.9, \Rz:=-13), v200, z200, Tooldata_9;
MoveJ RelTool (starting_position, 206,-52, 90.6 \Rx:=14.6, \Ry:=9.9, \Rz:=-13), v200, z200, Tooldata_9;
MoveJ RelTool (starting_position, 208,-52, 87.5 \Rx:=14.6, \Ry:=10.2, \Rz:=-13), v200, z200, Tooldata_9;
MoveJ RelTool (starting_position, 209,-56, 83.9 \Rx:=14.6, \Ry:=10.2, \Rz:=-14), v200, z200, Tooldata_9;
MoveJ RelTool (starting_position, 209,-56, 79.7 \Rx:=14.6, \Ry:=10.2, \Rz:=-14), v200, z200, Tooldata_9;
MoveJ RelTool (starting_position, 209,-56, 74.6 \Rx:=14.6, \Ry:=10.2, \Rz:=-14), v200, z200, Tooldata_9;
MoveJ RelTool (starting_position, 209,-56, 68.6 \Rx:=14.6, \Ry:=10.2, \Rz:=-14), v200, z200, Tooldata_9;
MoveJ RelTool (starting_position, 208,-56, 61.6 \Rx:=14.6, \Ry:=10.2, \Rz:=-14), v200, z200, Tooldata_9;
MoveJ RelTool (starting_position, 207,-56, 53.7 \Rx:=14.6, \Ry:=9.9, \Rz:=-14), v200, z200, Tooldata_9;
MoveJ RelTool (starting_position, 205,-56, 45.3 \Rx:=14.6, \Ry:=9.9, \Rz:=-14), v200, z200, Tooldata_9;
MoveJ RelTool (starting_position, 203,-56, 36.6 \Rx:=14.6, \Ry:=9.6, \Rz:=-14), v200, z200, Tooldata_9;
MoveJ RelTool (starting_position, 200,-56, 28 \Rx:=14.6, \Ry:=9.3, \Rz:=-14), v200, z200, Tooldata_9;
MoveJ RelTool (starting_position, 197,-56, 20.3 \Rx:=14.5, \Ry:=9, \Rz:=-14), v200, z200, Tooldata_9;
MoveJ RelTool (starting_position, 193,-56, 14.1 \Rx:=14.5, \Ry:=8.7, \Rz:=-14), v200, z200, Tooldata_9;
MoveJ RelTool (starting_position, 190,-56, 10 \Rx:=14.5, \Ry:=8.4, \Rz:=-14), v200, z200, Tooldata_9;
MoveJ RelTool (starting_position, 186,-56, 8.4 \Rx:=14.5, \Ry:=8.1, \Rz:=-14), v200, z200, Tooldata_9;
MoveJ RelTool (starting_position, 181,-56, 9.3 \Rx:=14.4, \Ry:=7.5, \Rz:=-14), v200, z200, Tooldata_9;
MoveJ RelTool (starting_position, 177,-56, 12.8 \Rx:=14.4, \Ry:=7.2, \Rz:=-14), v200, z200, Tooldata_9;
MoveJ RelTool (starting_position, 172,-56, 18.5 \Rx:=14.3, \Ry:=6.9, \Rz:=-14), v200, z200, Tooldata_9;
MoveJ RelTool (starting_position, 167,-56, 25.6 \Rx:=14.2, \Ry:=6.3, \Rz:=-14), v200, z200, Tooldata_9;
MoveJ RelTool (starting_position, 161,-56, 33.4 \Rx:=14.2, \Ry:=5.7, \Rz:=-14), v200, z200, Tooldata_9;
MoveJ RelTool (starting_position, 156,-56, 41.3 \Rx:=14.1, \Ry:=5.4, \Rz:=-14), v200, z200, Tooldata_9;
MoveJ RelTool (starting_position, 150,-56, 48.7 \Rx:=14, \Ry:=4.8, \Rz:=-14), v200, z200, Tooldata_9;
MoveJ RelTool (starting_position, 144,-56, 54.7 \Rx:=13.9, \Ry:=4.5, \Rz:=-14), v200, z200, Tooldata_9;
MoveJ RelTool (starting_position, 139,-56, 58.9 \Rx:=13.8, \Ry:=3.9, \Rz:=-14), v200, z200, Tooldata_9;
MoveJ RelTool (starting_position, 133,-56, 61.1 \Rx:=13.7, \Ry:=3.3, \Rz:=-14), v200, z200, Tooldata_9;
MoveJ RelTool (starting_position, 127,-56, 61.2 \Rx:=13.6, \Ry:=2.7, \Rz:=-14), v200, z200, Tooldata_9;
MoveJ RelTool (starting_position, 121,-56, 59.1 \Rx:=13.5, \Ry:=2.1, \Rz:=-14), v200, z200, Tooldata_9;
MoveJ RelTool (starting_position, 115,-56, 54.9 \Rx:=13.4, \Ry:=1.5, \Rz:=-14), v200, z200, Tooldata_9;
MoveJ RelTool (starting_position, 110,-56, 49 \Rx:=13.3, \Ry:=1.2, \Rz:=-14), v200, z200, Tooldata_9;
MoveJ RelTool (starting_position, 104,-56, 42 \Rx:=13.2, \Ry:=0.6, \Rz:=-14), v200, z200, Tooldata_9;
MoveJ RelTool (starting_position, 99,-56, 34.2 \Rx:=13.1, \Ry:=0.3, \Rz:=-14), v200, z200, Tooldata_9;
MoveJ RelTool (starting_position, 94,-56, 26.1 \Rx:=12.9, \Ry:=-0.3, \Rz:=-14), v200, z200, Tooldata_9;
MoveJ RelTool (starting_position, 89,-56, 18.3 \Rx:=12.8, \Ry:=-0.6, \Rz:=-14), v200, z200, Tooldata_9;
MoveJ RelTool (starting_position, 85,-56, 11.5 \Rx:=12.6, \Ry:=-0.9, \Rz:=-14), v200, z200, Tooldata_9;
MoveJ RelTool (starting_position, 80,-56, 6.3 \Rx:=12.5, \Ry:=-1.5, \Rz:=-14), v200, z200, Tooldata_9;
MoveJ RelTool (starting_position, 76,-56, 3.1 \Rx:=12.3, \Ry:=-1.8, \Rz:=-14), v200, z200, Tooldata_9;
MoveJ RelTool (starting_position, 73,-56, 2.3 \Rx:=12.2, \Ry:=-2.1, \Rz:=-14), v200, z200, Tooldata_9;
MoveJ RelTool (starting_position, 70,-56, 4.2 \Rx:=12, \Ry:=-2.4, \Rz:=-14), v200, z200, Tooldata_9;
MoveJ RelTool (starting_position, 67,-56, 8.7 \Rx:=11.8, \Ry:=-2.7, \Rz:=-14), v200, z200, Tooldata_9;
MoveJ RelTool (starting_position, 65,-56, 15.4 \Rx:=11.6, \Ry:=-3, \Rz:=-14), v200, z200, Tooldata_9;
MoveJ RelTool (starting_position, 63,-60, 23.6 \Rx:=11.5, \Ry:=-3.3, \Rz:=-15), v200, z200, Tooldata_9;
MoveJ RelTool (starting_position, 62,-60, 32.9 \Rx:=11.3, \Ry:=-3.3, \Rz:=-15), v200, z200, Tooldata_9;
MoveJ RelTool (starting_position, 61,-60, 42.6 \Rx:=11.1, \Ry:=-3.3, \Rz:=-15), v200, z200, Tooldata_9;
MoveJ RelTool (starting_position, 61,-60, 52.2 \Rx:=10.9, \Ry:=-3.3, \Rz:=-15), v200, z200, Tooldata_9;
MoveJ RelTool (starting_position, 62,-60, 61.2 \Rx:=10.7, \Ry:=-3.3, \Rz:=-15), v200, z200, Tooldata_9;
MoveJ RelTool (starting_position, 64,-60, 69.3 \Rx:=10.5, \Ry:=-3, \Rz:=-15), v200, z200, Tooldata_9;
MoveJ RelTool (starting_position, 66,-60, 76.4 \Rx:=10.3, \Ry:=-3, \Rz:=-15), v200, z200, Tooldata_9;
MoveJ RelTool (starting_position, 69,-60, 82.3 \Rx:=10.1, \Ry:=-2.7, \Rz:=-15), v200, z200, Tooldata_9;
MoveJ RelTool (starting_position, 73,-60, 87.2 \Rx:=9.9, \Ry:=-2.4, \Rz:=-15), v200, z200, Tooldata_9;
MoveJ RelTool (starting_position, 77,-60, 91 \Rx:=9.7, \Ry:=-1.8, \Rz:=-15), v200, z200, Tooldata_9;
MoveJ RelTool (starting_position, 82,-60, 93.8 \Rx:=9.5, \Ry:=-1.5, \Rz:=-15), v200, z200, Tooldata_9;
MoveJ RelTool (starting_position, 88,-60, 95.7 \Rx:=9.3, \Ry:=-0.9, \Rz:=-15), v200, z200, Tooldata_9;
MoveJ RelTool (starting_position, 94,-60, 97 \Rx:=9.1, \Ry:=-0.3, \Rz:=-15), v200, z200, Tooldata_9;
MoveJ RelTool (starting_position, 101,-60, 97.7 \Rx:=8.8, \Ry:=0.3, \Rz:=-15), v200, z200, Tooldata_9;
MoveJ RelTool (starting_position, 108,-60, 97.8 \Rx:=8.6, \Ry:=0.9, \Rz:=-15), v200, z200, Tooldata_9;
MoveJ RelTool (starting_position, 116,-60, 97.5 \Rx:=8.4, \Ry:=1.5, \Rz:=-15), v200, z200, Tooldata_9;
MoveJ RelTool (starting_position, 124,-60, 96.9 \Rx:=8.1, \Ry:=2.4, \Rz:=-15), v200, z200, Tooldata_9;
MoveJ RelTool (starting_position, 131,-60, 95.8 \Rx:=7.9, \Ry:=3.3, \Rz:=-15), v200, z200, Tooldata_9;
MoveJ RelTool (starting_position, 139,-60, 94.2 \Rx:=7.6, \Ry:=3.9, \Rz:=-15), v200, z200, Tooldata_9;
MoveJ RelTool (starting_position, 147,-60, 92.3 \Rx:=7.4, \Ry:=4.8, \Rz:=-15), v200, z200, Tooldata_9;
MoveJ RelTool (starting_position, 155,-60, 90 \Rx:=7.2, \Ry:=5.4, \Rz:=-15), v200, z200, Tooldata_9;
MoveJ RelTool (starting_position, 163,-60, 87.1 \Rx:=7, \Ry:=6, \Rz:=-15), v200, z200, Tooldata_9;
MoveJ RelTool (starting_position, 170,-60, 83.7 \Rx:=6.7, \Ry:=6.9, \Rz:=-15), v200, z200, Tooldata_9;
MoveJ RelTool (starting_position, 177,-60, 79.8 \Rx:=6.5, \Ry:=7.5, \Rz:=-15), v200, z200, Tooldata_9;
MoveJ RelTool (starting_position, 184,-60, 75.4 \Rx:=6.2, \Ry:=8.1, \Rz:=-15), v200, z200, Tooldata_9;
MoveJ RelTool (starting_position, 190,-60, 70.7 \Rx:=6, \Ry:=8.7, \Rz:=-15), v200, z200, Tooldata_9;
MoveJ RelTool (starting_position, 196,-60, 65.6 \Rx:=5.8, \Ry:=9, \Rz:=-15), v200, z200, Tooldata_9;
MoveJ RelTool (starting_position, 201,-60, 60.1 \Rx:=5.5, \Ry:=9.3, \Rz:=-15), v200, z200, Tooldata_9;
MoveJ RelTool (starting_position, 206,-60, 54.6 \Rx:=5.3, \Ry:=9.9, \Rz:=-15), v200, z200, Tooldata_9;
MoveJ RelTool (starting_position, 210,-60, 49.2 \Rx:=5.1, \Ry:=10.2, \Rz:=-15), v200, z200, Tooldata_9;
MoveJ RelTool (starting_position, 214,-60, 44.1 \Rx:=4.8, \Ry:=10.8, \Rz:=-15), v200, z200, Tooldata_9;
MoveJ RelTool (starting_position, 218,-60, 39.4 \Rx:=4.6, \Ry:=10.8, \Rz:=-15), v200, z200, Tooldata_9;
MoveJ RelTool (starting_position, 221,-60, 35.4 \Rx:=4.3, \Ry:=11.1, \Rz:=-15), v200, z200, Tooldata_9;
MoveJ RelTool (starting_position, 225,-60, 32.3 \Rx:=4.1, \Ry:=11.4, \Rz:=-15), v200, z200, Tooldata_9;
MoveJ RelTool (starting_position, 227,-60, 30.2 \Rx:=3.9, \Ry:=11.7, \Rz:=-15), v200, z200, Tooldata_9;
MoveJ RelTool (starting_position, 230,-60, 29.2 \Rx:=3.7, \Ry:=11.7, \Rz:=-15), v200, z200, Tooldata_9;
MoveJ RelTool (starting_position, 232,-60, 29.4 \Rx:=3.5, \Ry:=12, \Rz:=-15), v200, z200, Tooldata_9;
MoveJ RelTool (starting_position, 234,-60, 30.5 \Rx:=3.3, \Ry:=12.3, \Rz:=-15), v200, z200, Tooldata_9;
MoveJ RelTool (starting_position, 236,-60, 32.4 \Rx:=3.1, \Ry:=12.3, \Rz:=-15), v200, z200, Tooldata_9;
MoveJ RelTool (starting_position, 238,-60, 34.8 \Rx:=3, \Ry:=12.6, \Rz:=-15), v200, z200, Tooldata_9;
MoveJ RelTool (starting_position, 239,-60, 37.2 \Rx:=2.8, \Ry:=12.9, \Rz:=-15), v200, z200, Tooldata_9;
MoveJ RelTool (starting_position, 239,-60, 39.5 \Rx:=2.7, \Ry:=12.9, \Rz:=-15), v200, z200, Tooldata_9;
MoveJ RelTool (starting_position, 239,-60, 41.3 \Rx:=2.5, \Ry:=12.9, \Rz:=-15), v200, z200, Tooldata_9;
MoveJ RelTool (starting_position, 239,-60, 42.5 \Rx:=2.4, \Ry:=12.6, \Rz:=-15), v200, z200, Tooldata_9;
MoveJ RelTool (starting_position, 238,-60, 42.8 \Rx:=2.2, \Ry:=12.6, \Rz:=-15), v200, z200, Tooldata_9;
MoveJ RelTool (starting_position, 237,-60, 42.1 \Rx:=2.1, \Ry:=12.6, \Rz:=-15), v200, z200, Tooldata_9;
MoveJ RelTool (starting_position, 235,-60, 40.5 \Rx:=2, \Ry:=12.6, \Rz:=-15), v200, z200, Tooldata_9;
MoveJ RelTool (starting_position, 233,-60, 37.9 \Rx:=1.9, \Ry:=12.3, \Rz:=-15), v200, z200, Tooldata_9;
MoveJ RelTool (starting_position, 231,-60, 34.3 \Rx:=1.8, \Ry:=12, \Rz:=-15), v200, z200, Tooldata_9;
MoveJ RelTool (starting_position, 228,-60, 30 \Rx:=1.7, \Ry:=11.7, \Rz:=-15), v200, z200, Tooldata_9;
MoveJ RelTool (starting_position, 224,-60, 25 \Rx:=1.6, \Ry:=11.4, \Rz:=-15), v200, z200, Tooldata_9;
MoveJ RelTool (starting_position, 220,-60, 19.8 \Rx:=1.5, \Ry:=11.1, \Rz:=-15), v200, z200, Tooldata_9;
MoveJ RelTool (starting_position, 216,-60, 14.5 \Rx:=1.5, \Ry:=10.8, \Rz:=-15), v200, z200, Tooldata_9;
MoveJ RelTool (starting_position, 211,-60, 9.4 \Rx:=1.4, \Ry:=10.5, \Rz:=-15), v200, z200, Tooldata_9;
MoveJ RelTool (starting_position, 206,-60, 4.5 \Rx:=1.4, \Ry:=9.9, \Rz:=-15), v200, z200, Tooldata_9;
MoveJ RelTool (starting_position, 200,-60, 0.1 \Rx:=1.3, \Ry:=9.3, \Rz:=-15), v200, z200, Tooldata_9;
MoveJ RelTool (starting_position, 194,-60, -3.7 \Rx:=1.3, \Ry:=8.7, \Rz:=-15), v200, z200, Tooldata_9;
MoveJ RelTool (starting_position, 188,-60, -6.9 \Rx:=1.3, \Ry:=8.1, \Rz:=-15), v200, z200, Tooldata_9;
MoveJ RelTool (starting_position, 181,-60, -9.3 \Rx:=1.3, \Ry:=7.8, \Rz:=-15), v200, z200, Tooldata_9;
MoveJ RelTool (starting_position, 174,-60, -11.2 \Rx:=1.3, \Ry:=7.2, \Rz:=-15), v200, z200, Tooldata_9;
MoveJ RelTool (starting_position, 166,-60, -12.7 \Rx:=1.3, \Ry:=6.3, \Rz:=-15), v200, z200, Tooldata_9;
MoveJ RelTool (starting_position, 158,-60, -13.8 \Rx:=1.3, \Ry:=5.7, \Rz:=-15), v200, z200, Tooldata_9;
MoveJ RelTool (starting_position, 150,-60, -14.6 \Rx:=1.4, \Ry:=4.8, \Rz:=-15), v200, z200, Tooldata_9;
MoveJ RelTool (starting_position, 142,-60, -15.1 \Rx:=1.4, \Ry:=4.2, \Rz:=-15), v200, z200, Tooldata_9;
MoveJ RelTool (starting_position, 133,-60, -15.5 \Rx:=1.4, \Ry:=3.3, \Rz:=-15), v200, z200, Tooldata_9;
MoveJ RelTool (starting_position, 124,-60, -15.9 \Rx:=1.5, \Ry:=2.7, \Rz:=-15), v200, z200, Tooldata_9;
MoveJ RelTool (starting_position, 115,-60, -16.2 \Rx:=1.5, \Ry:=1.8, \Rz:=-15), v200, z200, Tooldata_9;
MoveJ RelTool (starting_position, 106,-60, -16.6 \Rx:=1.6, \Ry:=0.9, \Rz:=-15), v200, z200, Tooldata_9;
MoveJ RelTool (starting_position, 96,-60, -17.1 \Rx:=1.7, \Ry:=0.3, \Rz:=-15), v200, z200, Tooldata_9;
MoveJ RelTool (starting_position, 87,-60, -17.7 \Rx:=1.8, \Ry:=-0.6, \Rz:=-15), v200, z200, Tooldata_9;
MoveJ RelTool (starting_position, 77,-60, -18.5 \Rx:=1.9, \Ry:=-1.5, \Rz:=-15), v200, z200, Tooldata_9;
MoveJ RelTool (starting_position, 68,-60, -19.3 \Rx:=2, \Ry:=-2.4, \Rz:=-15), v200, z200, Tooldata_9;
MoveJ RelTool (starting_position, 58,-60, -20 \Rx:=2.1, \Ry:=-3.3, \Rz:=-15), v200, z200, Tooldata_9;
MoveJ RelTool (starting_position, 48,-60, -20.5 \Rx:=2.2, \Ry:=-4.2, \Rz:=-15), v200, z200, Tooldata_9;
MoveJ RelTool (starting_position, 39,-60, -20.7 \Rx:=2.3, \Ry:=-4.8, \Rz:=-15), v200, z200, Tooldata_9;
